// SIMATIC S7-200 SMART project (STEP 7-Micro/WIN SMART), CPU ST60

SYMBOL_TABLE Screen
X_JOG_Add_Scr    V1000.0  // X轴向上缓动按钮
X_JOG_Sub_Scr    V1000.1  // X轴向下缓动按钮
Y_JOG_Add_Scr    V1000.2
Y_JOG_Sub_Scr    V1000.3
Z_JOG_Up_Scr     V1000.4
Z_JOG_Dn_Scr     V1000.5
Teach_Btn_Setting V1000.6  // 教读设置按钮
Stop_Btn_Setting V1000.7  // 停止设置按钮
Home_Btn_Setting V1001.0  // 回原点按钮
Save_Btn_Setting V1001.1
X_Enable_Btn_Scr V1001.2
Y_Enable_Btn_Scr V1001.3
Z_Enable_Btn_Scr V1001.4
Speed_SW         V1001.5  // 速度状态指示位
Brake_Btn        V1001.6  // 刹车按钮
Clamp_Btn        V1001.7
Exit_Setting     V1005.7
Home_Lamp_Setting V1006.0  // X轴原点位指示灯
Teach_Lamp_Setting V1006.1  // 教读指示灯设置
Home_Btn_Manual  V1010.0
Stop_Btn_Manual  V1010.1
Teach_Btn_Manual V1010.2
Sholder1_Btn_Manual V1010.3
Select_Speed_Btn V1010.4  // 速度选择按钮
Sholder2_Btn_Manual V1010.5
Sholder3_Btn_Manual V1010.6
Exit_Btn_Manual  V1014.7
Home_Lamp_Manual V1015.0
Teach_Lamp_Manual V1015.1
Solder_Lamp      V1015.2
Start_Btn_Scr    V1020.0  // 屏幕运行按钮
Stop_Btn_Scr     V1020.1  // 屏幕停止按钮
Reset_Btn_Scr    V1020.2  // 复位屏幕按钮
Menu_Btn_Scr     V1020.3
Exit_MainMenu    V1020.4
Manual_Btn_Menu  V1020.5
ParaSet_Menu     V1020.6
Run_Lamp_Auto    V1021.0  // 自动运行指示灯
Stop_Lamp_Auto   V1021.1  // 自动停止指示灯
Reset_Lamp_Auto  V1021.2  // 自动复位指示灯
Run_Lamp_Blink   V1021.3
Stop_Lamp_Blink  V1021.4
Reset_Lamp_Blink V1021.5
Clr_Alarm_Btn    V1050.0
Call_Auto        V1150.0
Call_Manual      V1150.1
Call_Setting     V1150.2
Call_Solder1     V1150.3
Call_Solder2     V1150.4
Call_Solder3     V1150.5
HintTip_Stop     V1201.0  // 提示停止信息
HintTip_Reseting V1201.1  // 提示复位信息
HintTip_Running  V1201.2  // 提示运行信息
HintTip_Alarm    V1201.3  // 提示警报信息
HintTip_Ready    V1201.4  // 提示就绪信息
HintTip_Stopping V1201.5  // 提示停止信息
HintTip_Reseting1 V1201.6
X_Plus_Limit_Alarm V1501.0
X_Sub_Limit_Alarm V1501.1
Y_Plus_Limit_Alarm V1501.2
Y_Sub_Limit_Alarm V1501.3
Z_Up_Limit_Alarm V1501.4
Z_Dn_Limit_Alarm V1501.5
Clamp_At_Open_Alarm V1501.6
Clamp_At_Close_Alarm V1501.7
X_Curr_Pos_Scr   VD1900   // 屏幕X马达当前运行位置
Y_Curr_Pos_Scr   VD1904   // 屏幕Y马达当前运行位置
Z_Curr_Pos_Scr   VD1908   // 屏幕Z马达当前运行位置
X_High_Speed_Set VD4954   // X马达高速设置
X_Low_Speed_Set  VD4958   // X马达低速设置
Y_High_Speed_Set VD4962
Y_Low_Speed_Set  VD4966
Z_High_Speed_Set VD4970
Z_Low_Speed_Set  VD4974
X_Run_Speed_Set  VD4978   // X马达运行速度设置
Y_Run_Speed_Set  VD4982   // Y马达运行速度设置
Z_Run_Speed_Set  VD4986   // Z马达运行速度设置
X_POS1           VD5000
Y_POS1           VD6000
Z_POS1           VD7000
Cycle_Time       VW1100   // 单个循环周期
Choice_Aixs      VW1110
RunTip           VW1200
AlarmVar         VW1500
Screen_SW        VW1800
TotalPosNum_Set  VW4950   // 设置总的位置数值
Solder_Time      VW4952
Curr_PosNo_Scr   VW4990   // 屏幕当前XYZ马达运行位置数
Cycle_Counter    VW4992   // 循环计数器
END_SYMBOL_TABLE

SYMBOL_TABLE 系统符号
Always_On        SM0.0    // 始终接通
First_Scan_On    SM0.1    // 仅在第一个扫描周期时接通
Clock_1s         SM0.5    // 针对 1 s 的周期时间，时钟脉冲接通 0.5 s，断开 0.5 s。
P0_Config        SMB30    // 组态端口 0 通信：奇偶校验、每个字符的数据位数、波特率和协议
P0_Ctrl_Rcv      SMB87    // 接收消息控制
P0_End_Char      SMB89    // 消息结束字符
P0_Idle_Time     SMW90    // 给定的空行时间周期（以毫秒为单位）
P0_Timeout       SMW92    // 给定的字符间/消息定时器超时值（以毫秒为单位）
P0_Max_Char      SMB94    // 要接收的最大字符数（1 到 255 个字节）
END_SYMBOL_TABLE

SYMBOL_TABLE MotorStatus
X_Busy           M0.0
X_Curr_Dir       M0.1
Y_Busy           M0.2
Y_Curr_Dir       M0.3
Z_Busy           M0.4
Z_Curr_Dir       M0.5
X_Error_Code     MB1      // X马达错误代码
Y_Error_Code     MB2      // Y马达错误代码
Z_Error_Code     MB3      // Z马达运行错误代码
X_Curr_Speed     MD4      // X马达当前运行速度
Y_Curr_Speed     MD8      // Y马达当前运行速度
Z_Curr_Speed     MD12     // Z马达当前运行速度
END_SYMBOL_TABLE

SYMBOL_TABLE Machine
SpeedChoice_Pulse M18.0    // 速度选择脉冲
X_Home_EN        M18.1    // X轴归位使能信号状态位
Y_Home_EN        M18.2
Z_Home_EN        M18.3
X_Home_OK        M18.4
Y_Home_OK        M18.5
Z_Home_OK        M18.6    // Z轴准备就绪
X_Teach_EN       M18.7    // X马达教读使能
Y_Teach_EN       M19.0    // Y马达教读使能
Z_Teach_EN       M19.1    // Z马达教读使能
X_JOG_DIR        M19.2    // X轴缓动方向
Y_JOG_DIR        M19.3
Z_JOG_DIR        M19.4
X_JOG_EN         M19.5    // X轴缓动使能
Y_JOG_EN         M19.6
Z_JOG_EN         M19.7
Interlock_Manual M20.0
Interlock_Setting M20.1    // 自锁设置
X_Stop_Cmd       M20.2    // X马达停止指令
Y_Stop_Cmd       M20.3    // Y马达停止指令
Z_Stop_Cmd       M20.4    // Z马达停止指令
Motor_Ready      M20.5    // 马达就绪
XYZ_ORG_Cmd3     M22.0
XYZ_Home_OK      M20.6    // XYZ归位信号状态位
Z_Goto_UpPos     M20.7    // Z轴上升到最高位信号状态位
Init_MC_Sys      M21.0
XYZ_ORG_Cmd1     M21.6
XYZ_ORG_Cmd      M21.1    // XYZ归位起始位指令
Release_Brake_Step M21.2
Solder2_Cmd      M21.4
Solder3_Cmd      M21.5
Solder1_Cmd      M21.3
Step1_Auto_Lock  M25.0    // 自动锁定step1
Step1_Auto       M25.1    // 自动step1
Step2_X_Auto     M25.2    // X轴自动step2
Step2_Y_Auto     M25.3    // Y轴自动step2
Step3_Auto       M25.4    // 自动step3
Step4_Auto       M25.5    // 自动step4
X_Cmd_Pos        VD2000   // X马达位置指令
Y_Cmd_Pos        VD2004   // Y马达位置指令
Z_Cmd_Pos        VD2008   // Z马达位置指令
X_Debug_Speed    VD2012   // X马达调试（运行）速度
Y_Debug_Speed    VD2016
Z_Debug_Speed    VD2020   // Z马达调试速度
Cycle_Timer      T50      // 循环计时器
Sholder_Timer    T35
Solder_timer     T36
Brake_Release_Timer T34
Z_Home2          M29.2
Z_Home3          M29.3
Z_Home1          M29.1
XYZ_ORG_Cmd2     M21.7
END_SYMBOL_TABLE

SYMBOL_TABLE INPUT
X_AXIS_ZP        I0.0     // X轴马达索引
Y_AXIS_ZP        I0.1     // Y轴马达索引
Z_AXIS_ZP        I0.2     // Z轴马达索引
X_AXIS_LMT_Plus  I0.3     // X轴马达正限
X_AXIS_LMT_Sub   I0.4     // X轴马达负限
X_AXIS_HOME      I0.5     // X轴马达原点
Y_AXIS_LMT_Plus  I0.6     // Y轴马达正限
Y_AXIS_LMT_Sub   I0.7     // Y轴马达负限
Y_AXIS_HOME      I1.0     // Y轴马达原点
Z_AXIS_LMT_Plus  I1.1     // Z轴马达正限
Z_AXIS_LMT_Sub   I1.2     // Z轴马达负限
Z_AXIS_HOME      I1.3     // Z轴马达原点
X_AXIS_INPOS     I1.4     // X轴位置完成
X_AXIS_READY     I1.5     // X轴准备信号
X_AXIS_ALARM     I1.6     // X轴报警信号
Y_AXIS_INPOS     I1.7     // Y轴位置完成
Y_AXIS_READY     I2.0     // Y轴准备信号
Y_AXIS_ALARM     I2.1     // Y轴报警信号
Z_AXIS_INPOS     I2.2     // Z轴位置完成
Z_AXIS_READY     I2.3     // Z轴准备信号
Z_AXIS_ALARM     I2.4     // Z轴报警信号
START_BUTTON     I2.5     // 启动按钮
STOP_BUTTON      I2.6     // 停止按钮
RESET_BUTTON     I2.7     // 复位按钮
CLAMP_AT_OPEN    I3.0     // 夹子打开感应
CLAMP_AT_CLOSE   I3.1     // 夹子关闭感应
END_SYMBOL_TABLE

SYMBOL_TABLE OUTPUT
X_AXIS_PULSE     Q0.0     // X轴脉冲信号
Y_AXIS_PULSE     Q0.1     // Y轴脉冲信号
X_AXIS_DIR       Q0.2     // X轴方向信号
Z_AXIS_PULSE     Q0.3     // Z轴脉冲信号
X_AXIS_ENABLE    Q0.4     // X轴使能信号
Y_AXIS_ENABLE    Q0.5     // Y轴使能信号
Z_AXIS_ENABLE    Q0.6     // Z轴使能信号
Y_AXIS_DIR       Q0.7     // Y轴方向信号
Z_AXIS_DIR       Q1.0     // Z轴方向信号
X_ALARM_CLEAR    Q1.1     // X轴报警清除
Y_ALARM_CLEAR    Q1.2     // Y轴报警清除
Z_ALARM_CLEAR    Q1.3     // Z轴报警清除
Z_BRAKE_RELEASE  Q1.4     // Z轴刹车释放
CLAMP_OPEN_VALVE Q1.5     // 夹打开阀
CLAMP_CLOSE_VALVE Q1.6     // 夹关闭阀
START_LAMP       Q2.0     // 启动指示灯
STOP_LAMP        Q2.1     // 停止指示灯
RESET_LAMP       Q2.2     // 复位指示灯
END_SYMBOL_TABLE

SYMBOL_TABLE Solder1
Step1_Solder1    M26.0
Step2_Solder1    M26.1
Step3_Solder1    M26.2
Step4_Solder1    M26.3
Step5_Solder1    M26.4
Step6_Solder1    M26.5
Step7_Solder1    M26.6
X_No_1           VD3000
X_No_2           VD3004
solder_No1       VW4998
END_SYMBOL_TABLE

SYMBOL_TABLE Solder3
Step1_Solder3    M27.3
Step2_Solder3    M27.4
Step3_Solder3    M27.5
Step4_Solder3    M27.6
Step5_Solder3    M27.7
Step6_Solder3    M28.0
Step7_Solder3    M28.1
Step8_Solder3    M28.2
END_SYMBOL_TABLE

SYMBOL_TABLE Solder2
Step1_Solder2    M28.3
Step2_Solder2    M28.4
Step3_Solder2    M26.7
Step4_Solder2    M27.0
Step5_Solder2    M27.1
Step6_Solder2    M27.2
Step7_Solder2    M28.5
Step8_Solder2    M28.6
END_SYMBOL_TABLE

ORGANIZATION_BLOCK 程序块:OB1
TITLE=程序注释
VAR
AutoScreen:WORD;	// LW0 
ManualScreen:WORD;	// LW2 
SettingScreen:WORD;	// LW4 
AlarmScreen:WORD;	// LW6 
MainScreen:WORD;	// LW8 
END_VAR
BEGIN
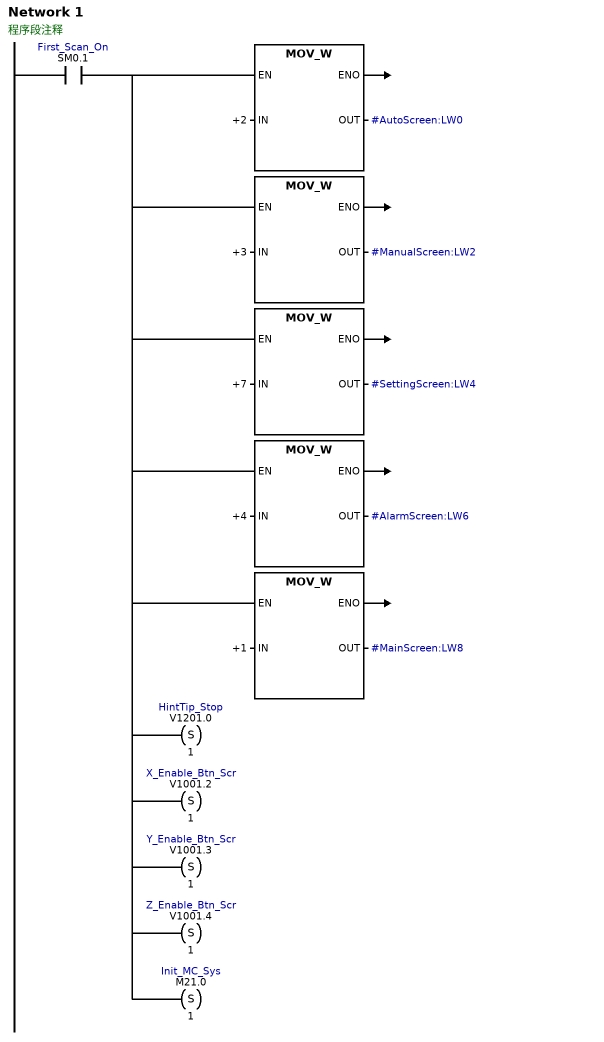
Network 1
// 程序段注释
LD     First_Scan_On:SM0.1
MOVW   +2, #AutoScreen:LW0
MOVW   +3, #ManualScreen:LW2
MOVW   +7, #SettingScreen:LW4
MOVW   +4, #AlarmScreen:LW6
MOVW   +1, #MainScreen:LW8
S      HintTip_Stop:V1201.0, 1
S      X_Enable_Btn_Scr:V1001.2, 1
S      Y_Enable_Btn_Scr:V1001.3, 1
S      Z_Enable_Btn_Scr:V1001.4, 1
S      Init_MC_Sys:M21.0, 1
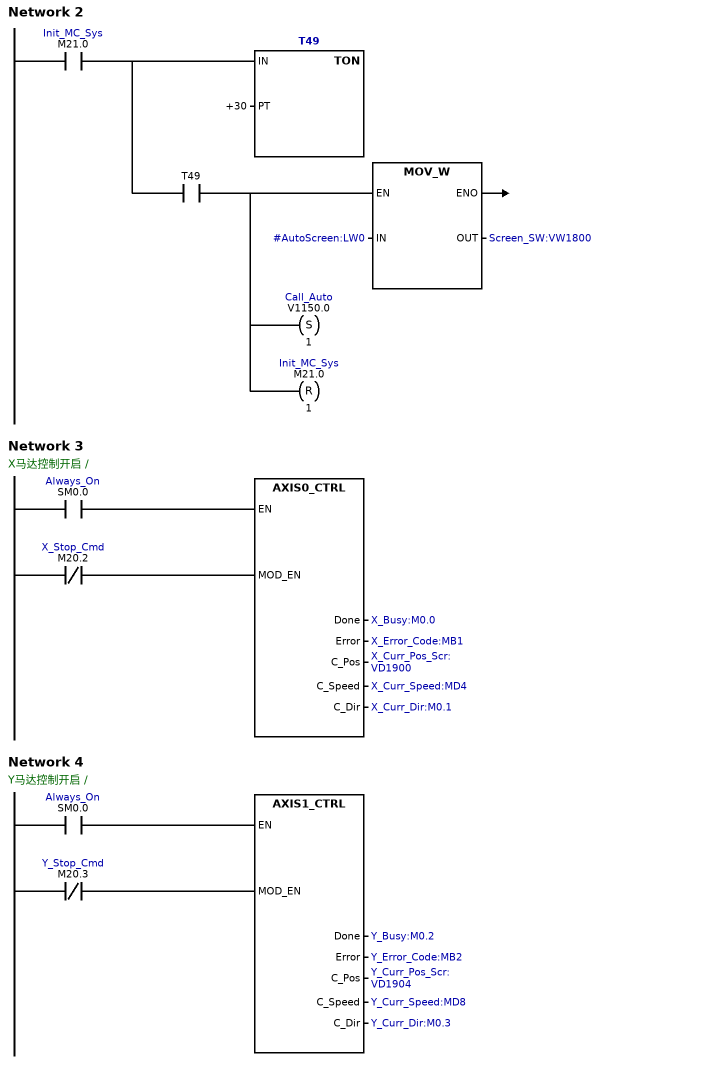
Network 2
LD     Init_MC_Sys:M21.0
TON    T49, +30
A      T49
MOVW   #AutoScreen:LW0, Screen_SW:VW1800
S      Call_Auto:V1150.0, 1
R      Init_MC_Sys:M21.0, 1
Network 3
// X马达控制开启
// 
LD     Always_On:SM0.0
=      L60.0
LDN    X_Stop_Cmd:M20.2
=      L63.7
LD     L60.0
CALL   AXIS0_CTRL:SBR1, L63.7, X_Busy:M0.0, X_Error_Code:MB1, X_Curr_Pos_Scr:VD1900, X_Curr_Speed:MD4, X_Curr_Dir:M0.1
Network 4
// Y马达控制开启
// 
LD     Always_On:SM0.0
=      L60.0
LDN    Y_Stop_Cmd:M20.3
=      L63.7
LD     L60.0
CALL   AXIS1_CTRL:SBR12, L63.7, Y_Busy:M0.2, Y_Error_Code:MB2, Y_Curr_Pos_Scr:VD1904, Y_Curr_Speed:MD8, Y_Curr_Dir:M0.3
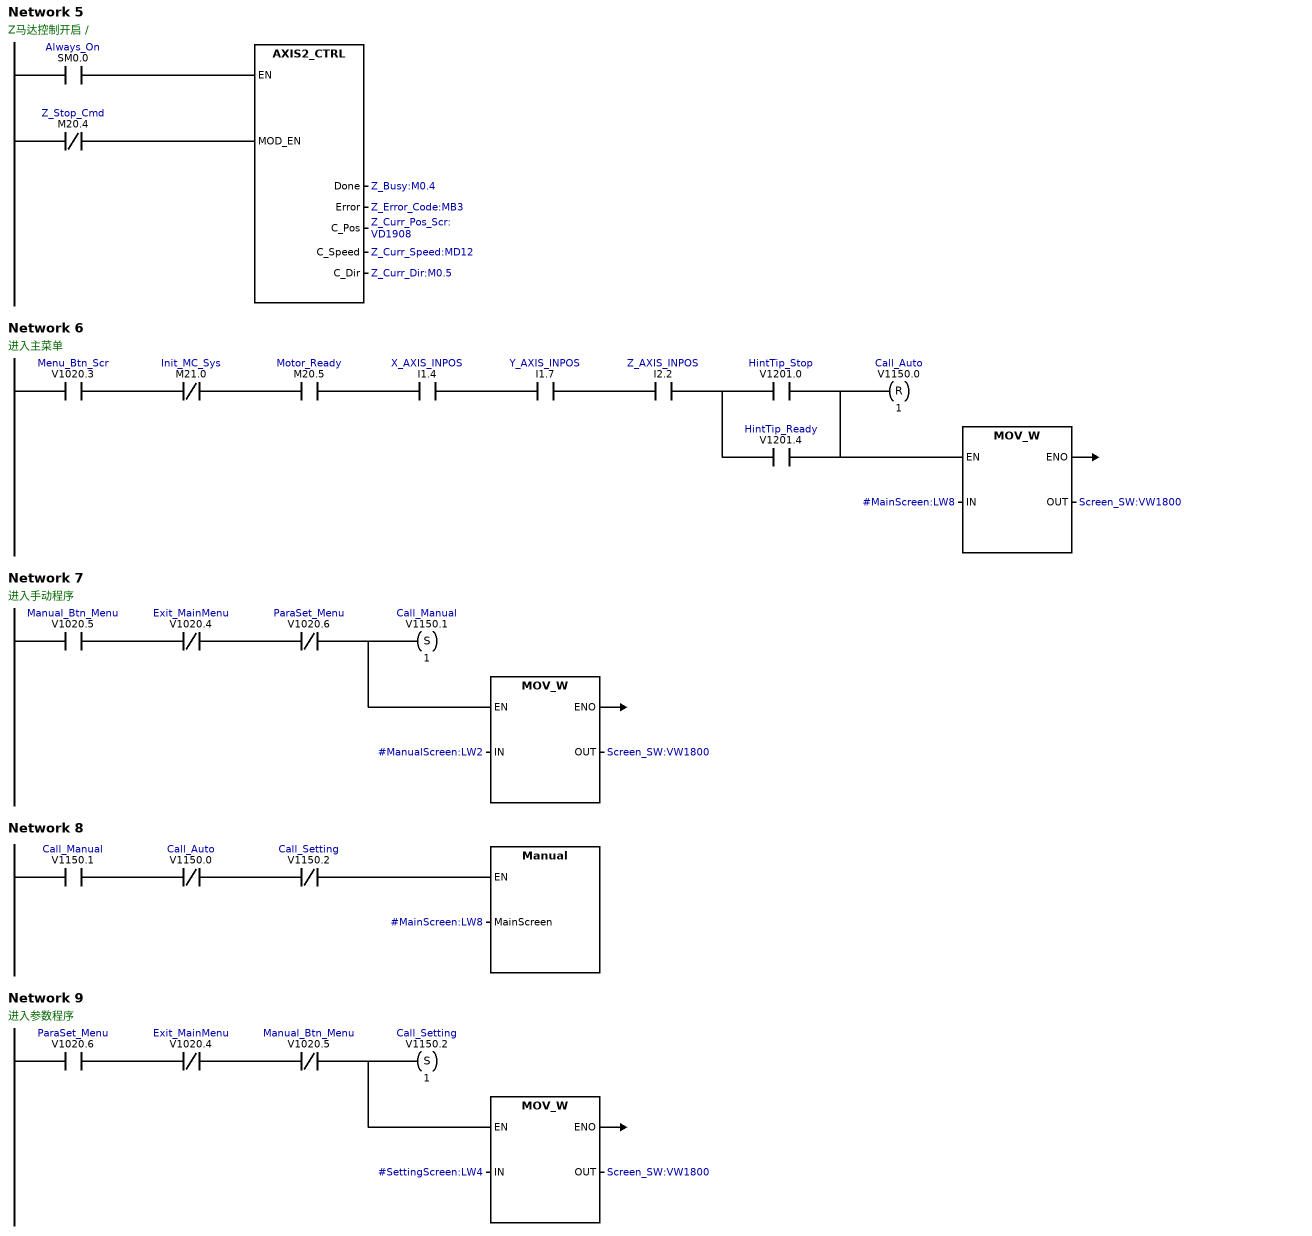
Network 5
// Z马达控制开启
// 
LD     Always_On:SM0.0
=      L60.0
LDN    Z_Stop_Cmd:M20.4
=      L63.7
LD     L60.0
CALL   AXIS2_CTRL:SBR23, L63.7, Z_Busy:M0.4, Z_Error_Code:MB3, Z_Curr_Pos_Scr:VD1908, Z_Curr_Speed:MD12, Z_Curr_Dir:M0.5
Network 6
// 进入主菜单
LD     Menu_Btn_Scr:V1020.3
AN     Init_MC_Sys:M21.0
A      Motor_Ready:M20.5
A      X_AXIS_INPOS:I1.4
A      Y_AXIS_INPOS:I1.7
A      Z_AXIS_INPOS:I2.2
LD     HintTip_Stop:V1201.0
O      HintTip_Ready:V1201.4
ALD
R      Call_Auto:V1150.0, 1
MOVW   #MainScreen:LW8, Screen_SW:VW1800
Network 7
// 进入手动程序
LD     Manual_Btn_Menu:V1020.5
AN     Exit_MainMenu:V1020.4
AN     ParaSet_Menu:V1020.6
S      Call_Manual:V1150.1, 1
MOVW   #ManualScreen:LW2, Screen_SW:VW1800
Network 8
LD     Call_Manual:V1150.1
AN     Call_Auto:V1150.0
AN     Call_Setting:V1150.2
CALL   Manual:SBR0, #MainScreen:LW8
Network 9
// 进入参数程序
LD     ParaSet_Menu:V1020.6
AN     Exit_MainMenu:V1020.4
AN     Manual_Btn_Menu:V1020.5
S      Call_Setting:V1150.2, 1
MOVW   #SettingScreen:LW4, Screen_SW:VW1800
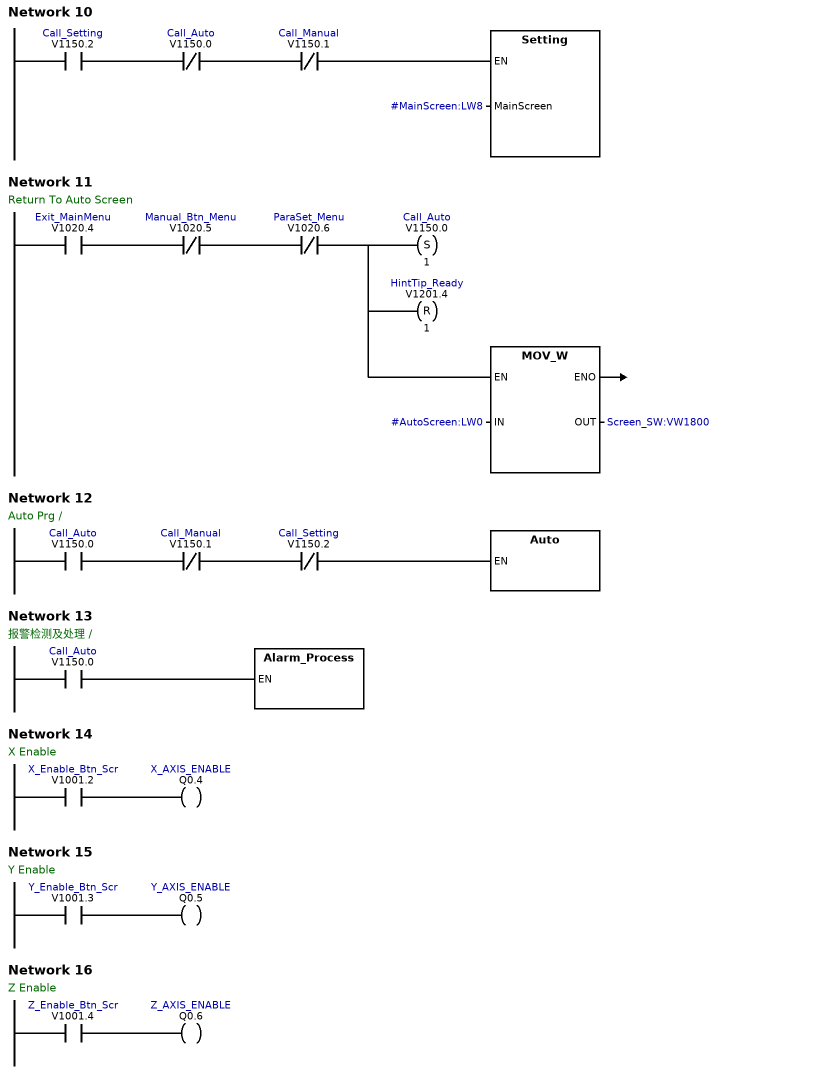
Network 10
LD     Call_Setting:V1150.2
AN     Call_Auto:V1150.0
AN     Call_Manual:V1150.1
CALL   Setting:SBR35, #MainScreen:LW8
Network 11
// Return To Auto Screen
LD     Exit_MainMenu:V1020.4
AN     Manual_Btn_Menu:V1020.5
AN     ParaSet_Menu:V1020.6
S      Call_Auto:V1150.0, 1
R      HintTip_Ready:V1201.4, 1
MOVW   #AutoScreen:LW0, Screen_SW:VW1800
Network 12
// Auto Prg
// 
LD     Call_Auto:V1150.0
AN     Call_Manual:V1150.1
AN     Call_Setting:V1150.2
CALL   Auto:SBR34
Network 13
// 报警检测及处理
// 
LD     Call_Auto:V1150.0
CALL   Alarm_Process:SBR36
Network 14
// X Enable
LD     X_Enable_Btn_Scr:V1001.2
=      X_AXIS_ENABLE:Q0.4
Network 15
// Y Enable
LD     Y_Enable_Btn_Scr:V1001.3
=      Y_AXIS_ENABLE:Q0.5
Network 16
// Z Enable
LD     Z_Enable_Btn_Scr:V1001.4
=      Z_AXIS_ENABLE:Q0.6
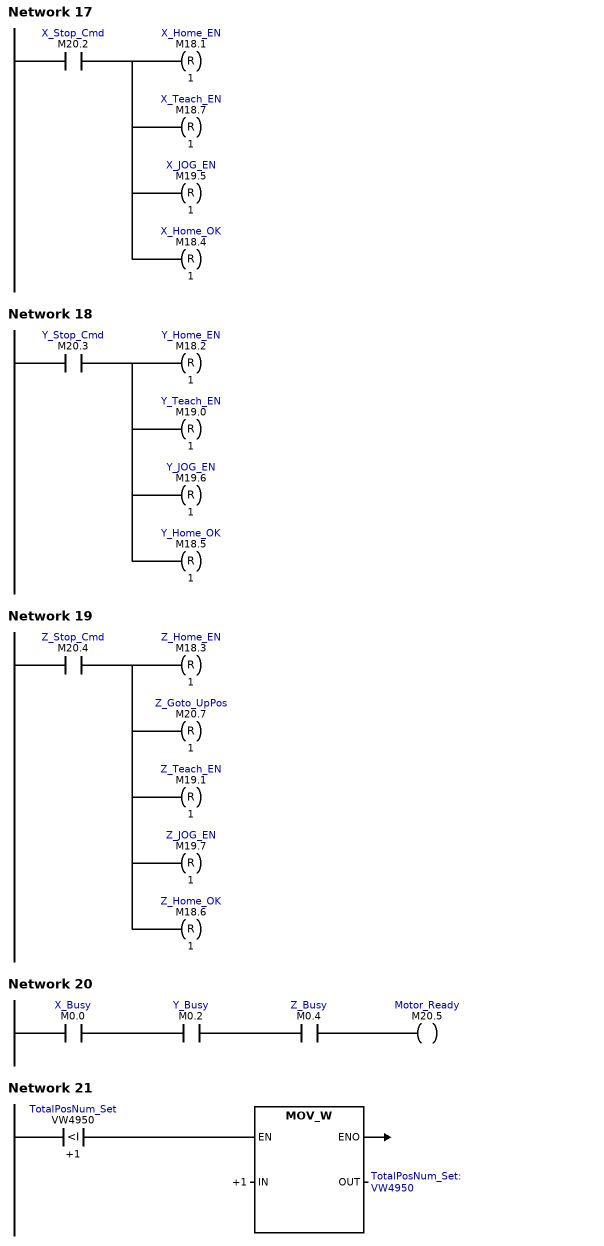
Network 17
LD     X_Stop_Cmd:M20.2
R      X_Home_EN:M18.1, 1
R      X_Teach_EN:M18.7, 1
R      X_JOG_EN:M19.5, 1
R      X_Home_OK:M18.4, 1
Network 18
LD     Y_Stop_Cmd:M20.3
R      Y_Home_EN:M18.2, 1
R      Y_Teach_EN:M19.0, 1
R      Y_JOG_EN:M19.6, 1
R      Y_Home_OK:M18.5, 1
Network 19
LD     Z_Stop_Cmd:M20.4
R      Z_Home_EN:M18.3, 1
R      Z_Goto_UpPos:M20.7, 1
R      Z_Teach_EN:M19.1, 1
R      Z_JOG_EN:M19.7, 1
R      Z_Home_OK:M18.6, 1
Network 20
LD     X_Busy:M0.0
A      Y_Busy:M0.2
A      Z_Busy:M0.4
=      Motor_Ready:M20.5
Network 21
LDW<   TotalPosNum_Set:VW4950, +1
MOVW   +1, TotalPosNum_Set:VW4950
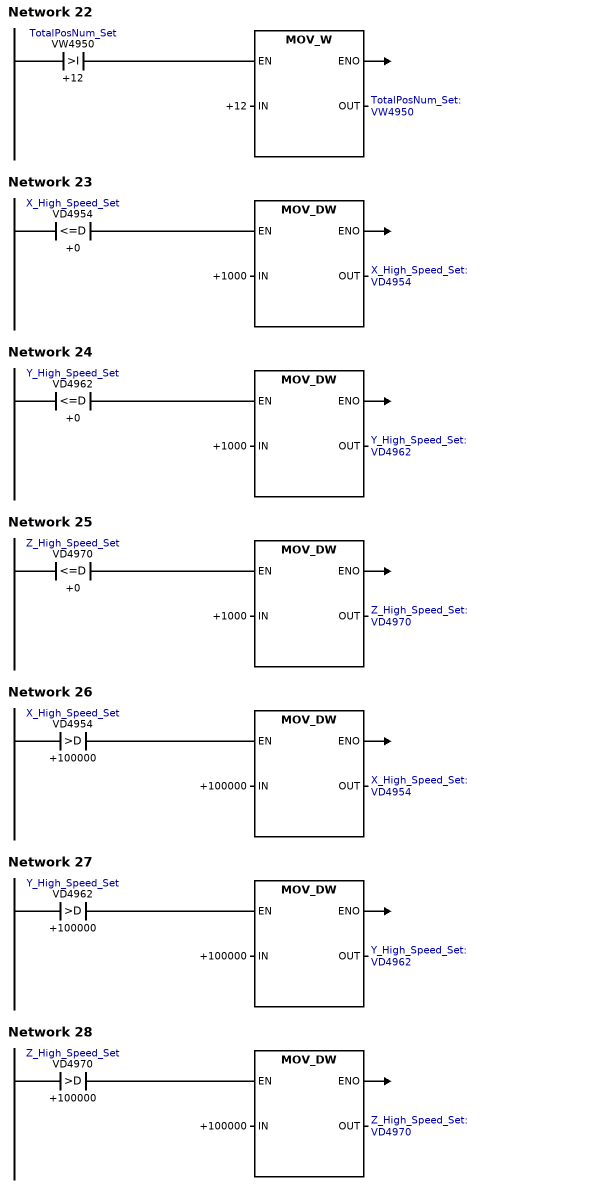
Network 22
LDW>   TotalPosNum_Set:VW4950, +12
MOVW   +12, TotalPosNum_Set:VW4950
Network 23
LDD<=  X_High_Speed_Set:VD4954, +0
MOVD   +1000, X_High_Speed_Set:VD4954
Network 24
LDD<=  Y_High_Speed_Set:VD4962, +0
MOVD   +1000, Y_High_Speed_Set:VD4962
Network 25
LDD<=  Z_High_Speed_Set:VD4970, +0
MOVD   +1000, Z_High_Speed_Set:VD4970
Network 26
LDD>   X_High_Speed_Set:VD4954, +100000
MOVD   +100000, X_High_Speed_Set:VD4954
Network 27
LDD>   Y_High_Speed_Set:VD4962, +100000
MOVD   +100000, Y_High_Speed_Set:VD4962
Network 28
LDD>   Z_High_Speed_Set:VD4970, +100000
MOVD   +100000, Z_High_Speed_Set:VD4970
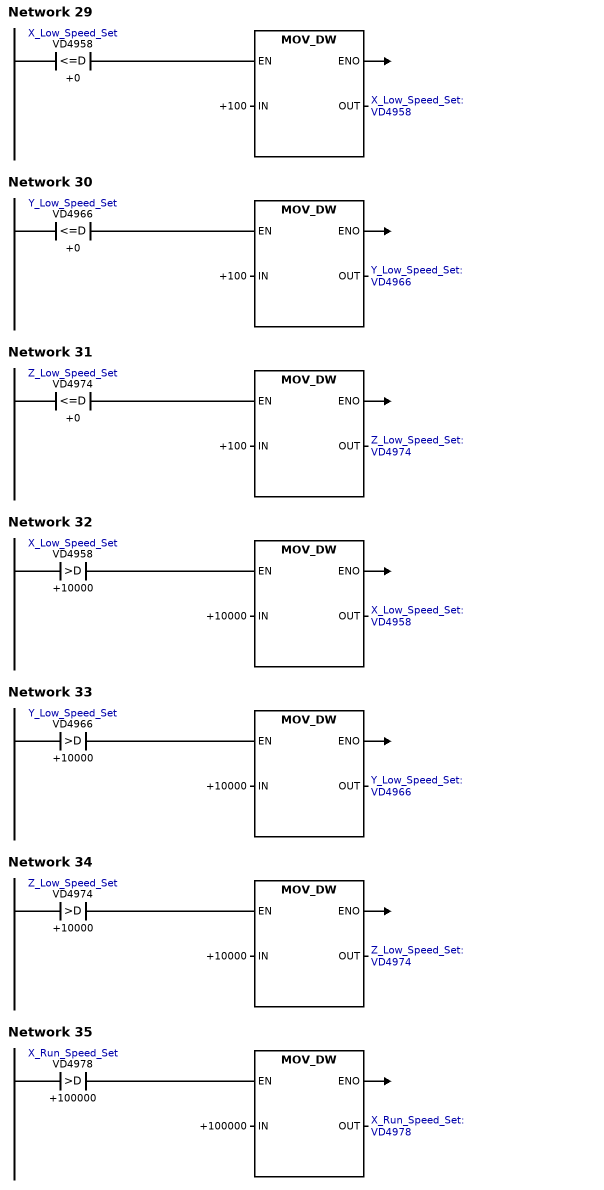
Network 29
LDD<=  X_Low_Speed_Set:VD4958, +0
MOVD   +100, X_Low_Speed_Set:VD4958
Network 30
LDD<=  Y_Low_Speed_Set:VD4966, +0
MOVD   +100, Y_Low_Speed_Set:VD4966
Network 31
LDD<=  Z_Low_Speed_Set:VD4974, +0
MOVD   +100, Z_Low_Speed_Set:VD4974
Network 32
LDD>   X_Low_Speed_Set:VD4958, +10000
MOVD   +10000, X_Low_Speed_Set:VD4958
Network 33
LDD>   Y_Low_Speed_Set:VD4966, +10000
MOVD   +10000, Y_Low_Speed_Set:VD4966
Network 34
LDD>   Z_Low_Speed_Set:VD4974, +10000
MOVD   +10000, Z_Low_Speed_Set:VD4974
Network 35
LDD>   X_Run_Speed_Set:VD4978, +100000
MOVD   +100000, X_Run_Speed_Set:VD4978
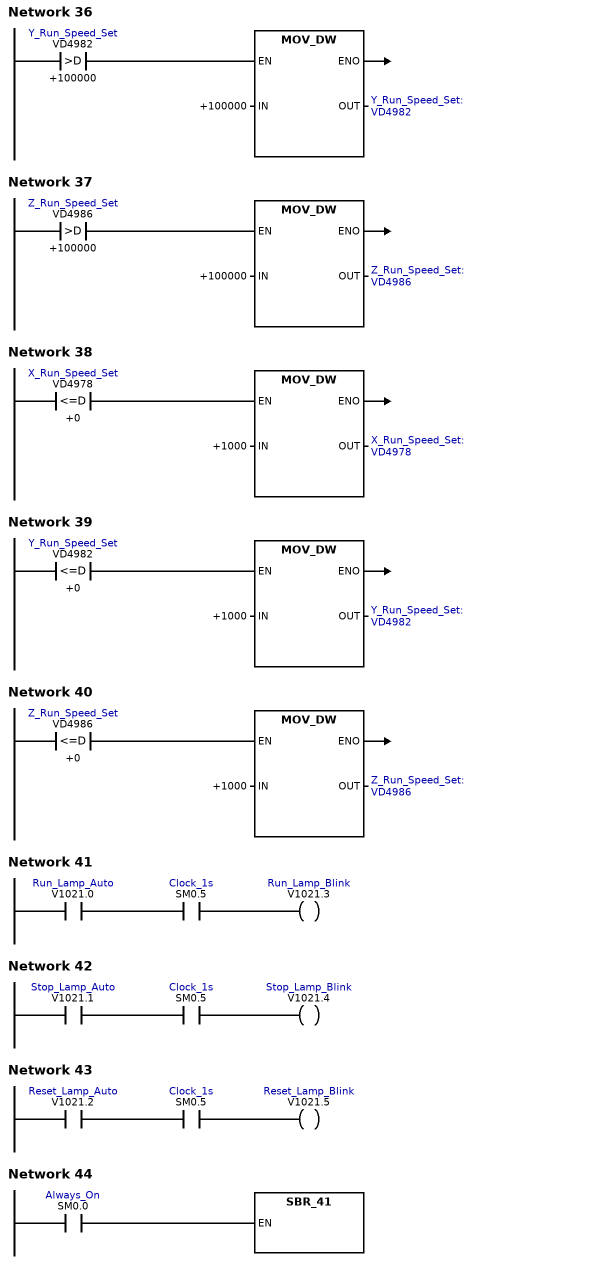
Network 36
LDD>   Y_Run_Speed_Set:VD4982, +100000
MOVD   +100000, Y_Run_Speed_Set:VD4982
Network 37
LDD>   Z_Run_Speed_Set:VD4986, +100000
MOVD   +100000, Z_Run_Speed_Set:VD4986
Network 38
LDD<=  X_Run_Speed_Set:VD4978, +0
MOVD   +1000, X_Run_Speed_Set:VD4978
Network 39
LDD<=  Y_Run_Speed_Set:VD4982, +0
MOVD   +1000, Y_Run_Speed_Set:VD4982
Network 40
LDD<=  Z_Run_Speed_Set:VD4986, +0
MOVD   +1000, Z_Run_Speed_Set:VD4986
Network 41
LD     Run_Lamp_Auto:V1021.0
A      Clock_1s:SM0.5
=      Run_Lamp_Blink:V1021.3
Network 42
LD     Stop_Lamp_Auto:V1021.1
A      Clock_1s:SM0.5
=      Stop_Lamp_Blink:V1021.4
Network 43
LD     Reset_Lamp_Auto:V1021.2
A      Clock_1s:SM0.5
=      Reset_Lamp_Blink:V1021.5
Network 44
LD     Always_On:SM0.0
CALL   SBR_41:SBR41
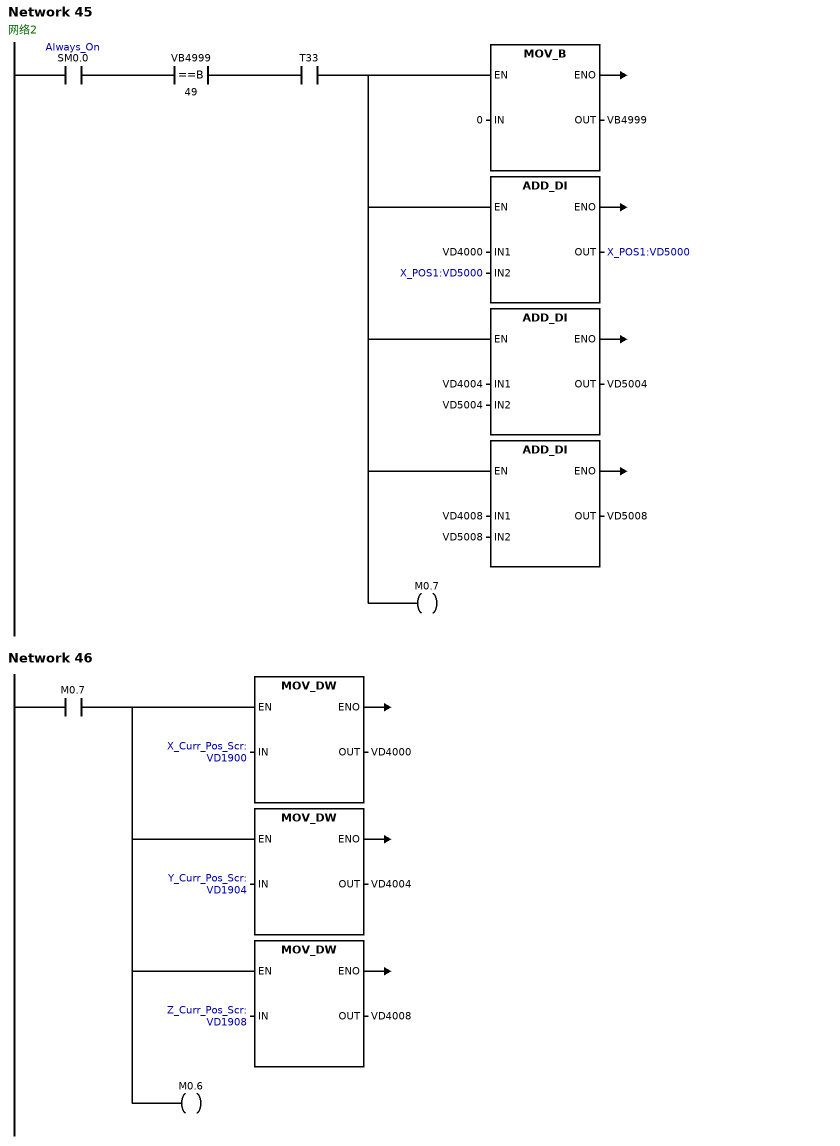
Network 45
// 网络2  
LD     Always_On:SM0.0
AB=    VB4999, 49
A      T33
MOVB   0, VB4999
+D     VD4000, X_POS1:VD5000
+D     VD4004, VD5004
+D     VD4008, VD5008
=      M0.7
Network 46
//   
LD     M0.7
MOVD   X_Curr_Pos_Scr:VD1900, VD4000
MOVD   Y_Curr_Pos_Scr:VD1904, VD4004
MOVD   Z_Curr_Pos_Scr:VD1908, VD4008
=      M0.6
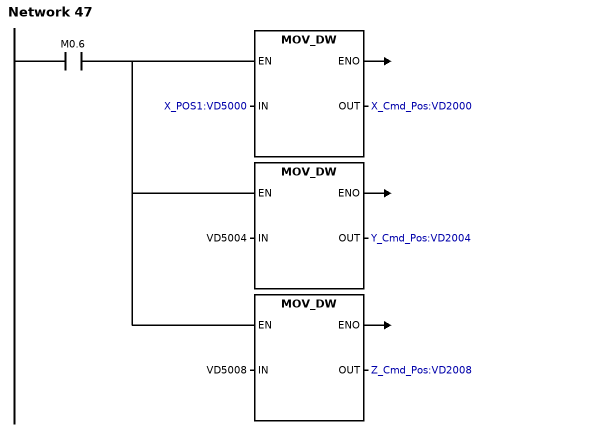
Network 47
LD     M0.6
MOVD   X_POS1:VD5000, X_Cmd_Pos:VD2000
MOVD   VD5004, Y_Cmd_Pos:VD2004
MOVD   VD5008, Z_Cmd_Pos:VD2008
END_ORGANIZATION_BLOCK

SUBROUTINE_BLOCK Manual:SBR0
TITLE=子例程注释
VAR_INPUT
MainScreen:WORD;	// LW0 
END_VAR
VAR
X_Home_Err:BYTE;	// LB2 
Y_Home_Err:BYTE;	// LB3 
Z_Home_Err:BYTE;	// LB4 
X_Teach_Done:BOOL;	// L5.0 
Y_Teach_Done:BOOL;	// L5.1 
Z_Teach_Done:BOOL;	// L5.2 
X_Teach_Err:BYTE;	// LB6 
Y_Teach_Err:BYTE;	// LB7 
Z_Teach_Err:BYTE;	// LB8 
X_JOG_ERR:BYTE;	// LB9 
Y_JOG_ERR:BYTE;	// LB10 
Z_JOG_ERR:BYTE;	// LB11 
X_Curr_Dir:BOOL;	// L12.0 
Y_Curr_Dir:BOOL;	// L12.1 
Z_Curr_Dir:BOOL;	// L12.2 
END_VAR
BEGIN
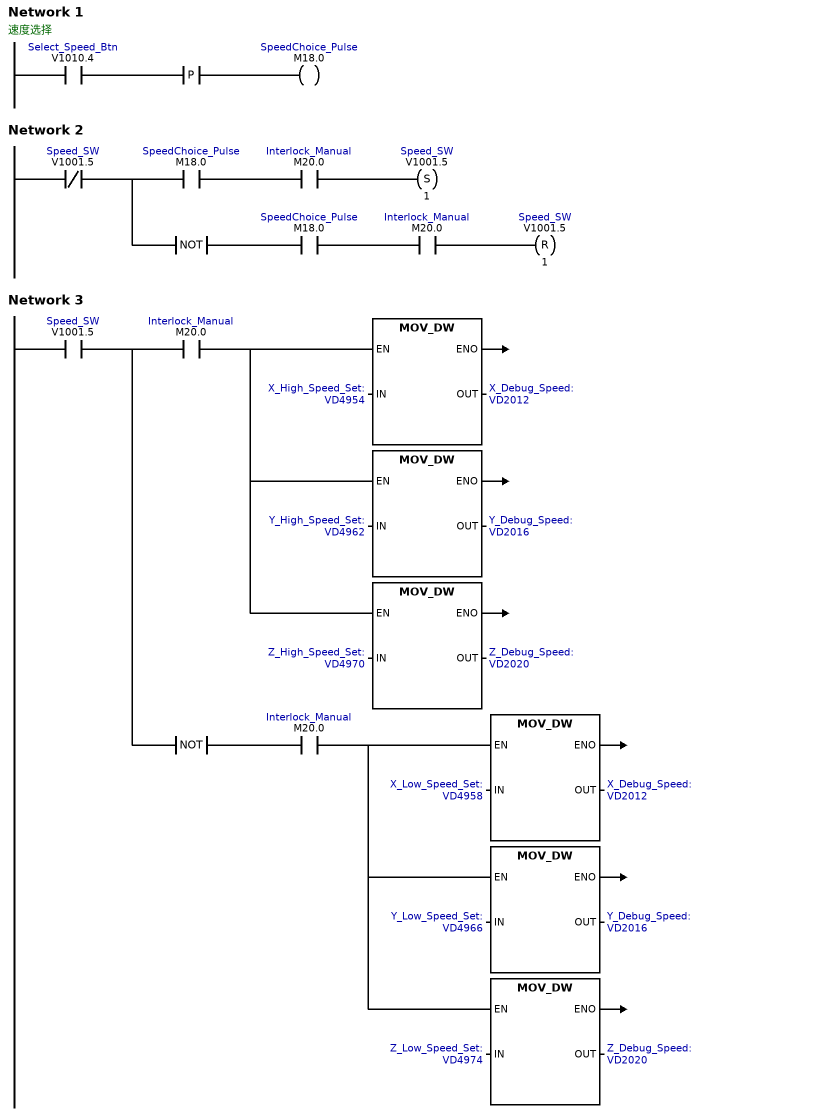
Network 1
// 速度选择
LD     Select_Speed_Btn:V1010.4
EU
=      SpeedChoice_Pulse:M18.0
Network 2
LDN    Speed_SW:V1001.5
LPS
A      SpeedChoice_Pulse:M18.0
A      Interlock_Manual:M20.0
S      Speed_SW:V1001.5, 1
LPP
NOT
A      SpeedChoice_Pulse:M18.0
A      Interlock_Manual:M20.0
R      Speed_SW:V1001.5, 1
Network 3
LD     Speed_SW:V1001.5
LPS
A      Interlock_Manual:M20.0
MOVD   X_High_Speed_Set:VD4954, X_Debug_Speed:VD2012
MOVD   Y_High_Speed_Set:VD4962, Y_Debug_Speed:VD2016
MOVD   Z_High_Speed_Set:VD4970, Z_Debug_Speed:VD2020
LPP
NOT
A      Interlock_Manual:M20.0
MOVD   X_Low_Speed_Set:VD4958, X_Debug_Speed:VD2012
MOVD   Y_Low_Speed_Set:VD4966, Y_Debug_Speed:VD2016
MOVD   Z_Low_Speed_Set:VD4974, Z_Debug_Speed:VD2020
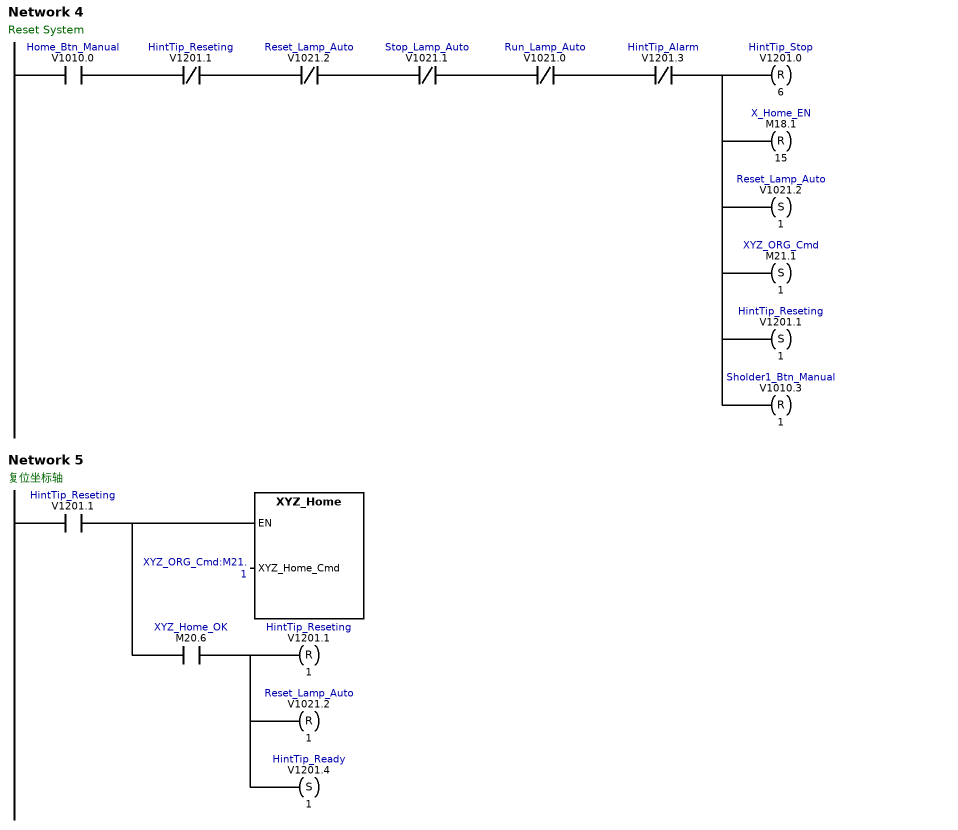
Network 4
// Reset System
LD     Home_Btn_Manual:V1010.0
AN     HintTip_Reseting:V1201.1
AN     Reset_Lamp_Auto:V1021.2
AN     Stop_Lamp_Auto:V1021.1
AN     Run_Lamp_Auto:V1021.0
AN     HintTip_Alarm:V1201.3
R      HintTip_Stop:V1201.0, 6
R      X_Home_EN:M18.1, 15
S      Reset_Lamp_Auto:V1021.2, 1
S      XYZ_ORG_Cmd:M21.1, 1
S      HintTip_Reseting:V1201.1, 1
R      Sholder1_Btn_Manual:V1010.3, 1
Network 5
// 复位坐标轴
LD     HintTip_Reseting:V1201.1
CALL   XYZ_Home:SBR37, XYZ_ORG_Cmd:M21.1
A      XYZ_Home_OK:M20.6
R      HintTip_Reseting:V1201.1, 1
R      Reset_Lamp_Auto:V1021.2, 1
S      HintTip_Ready:V1201.4, 1
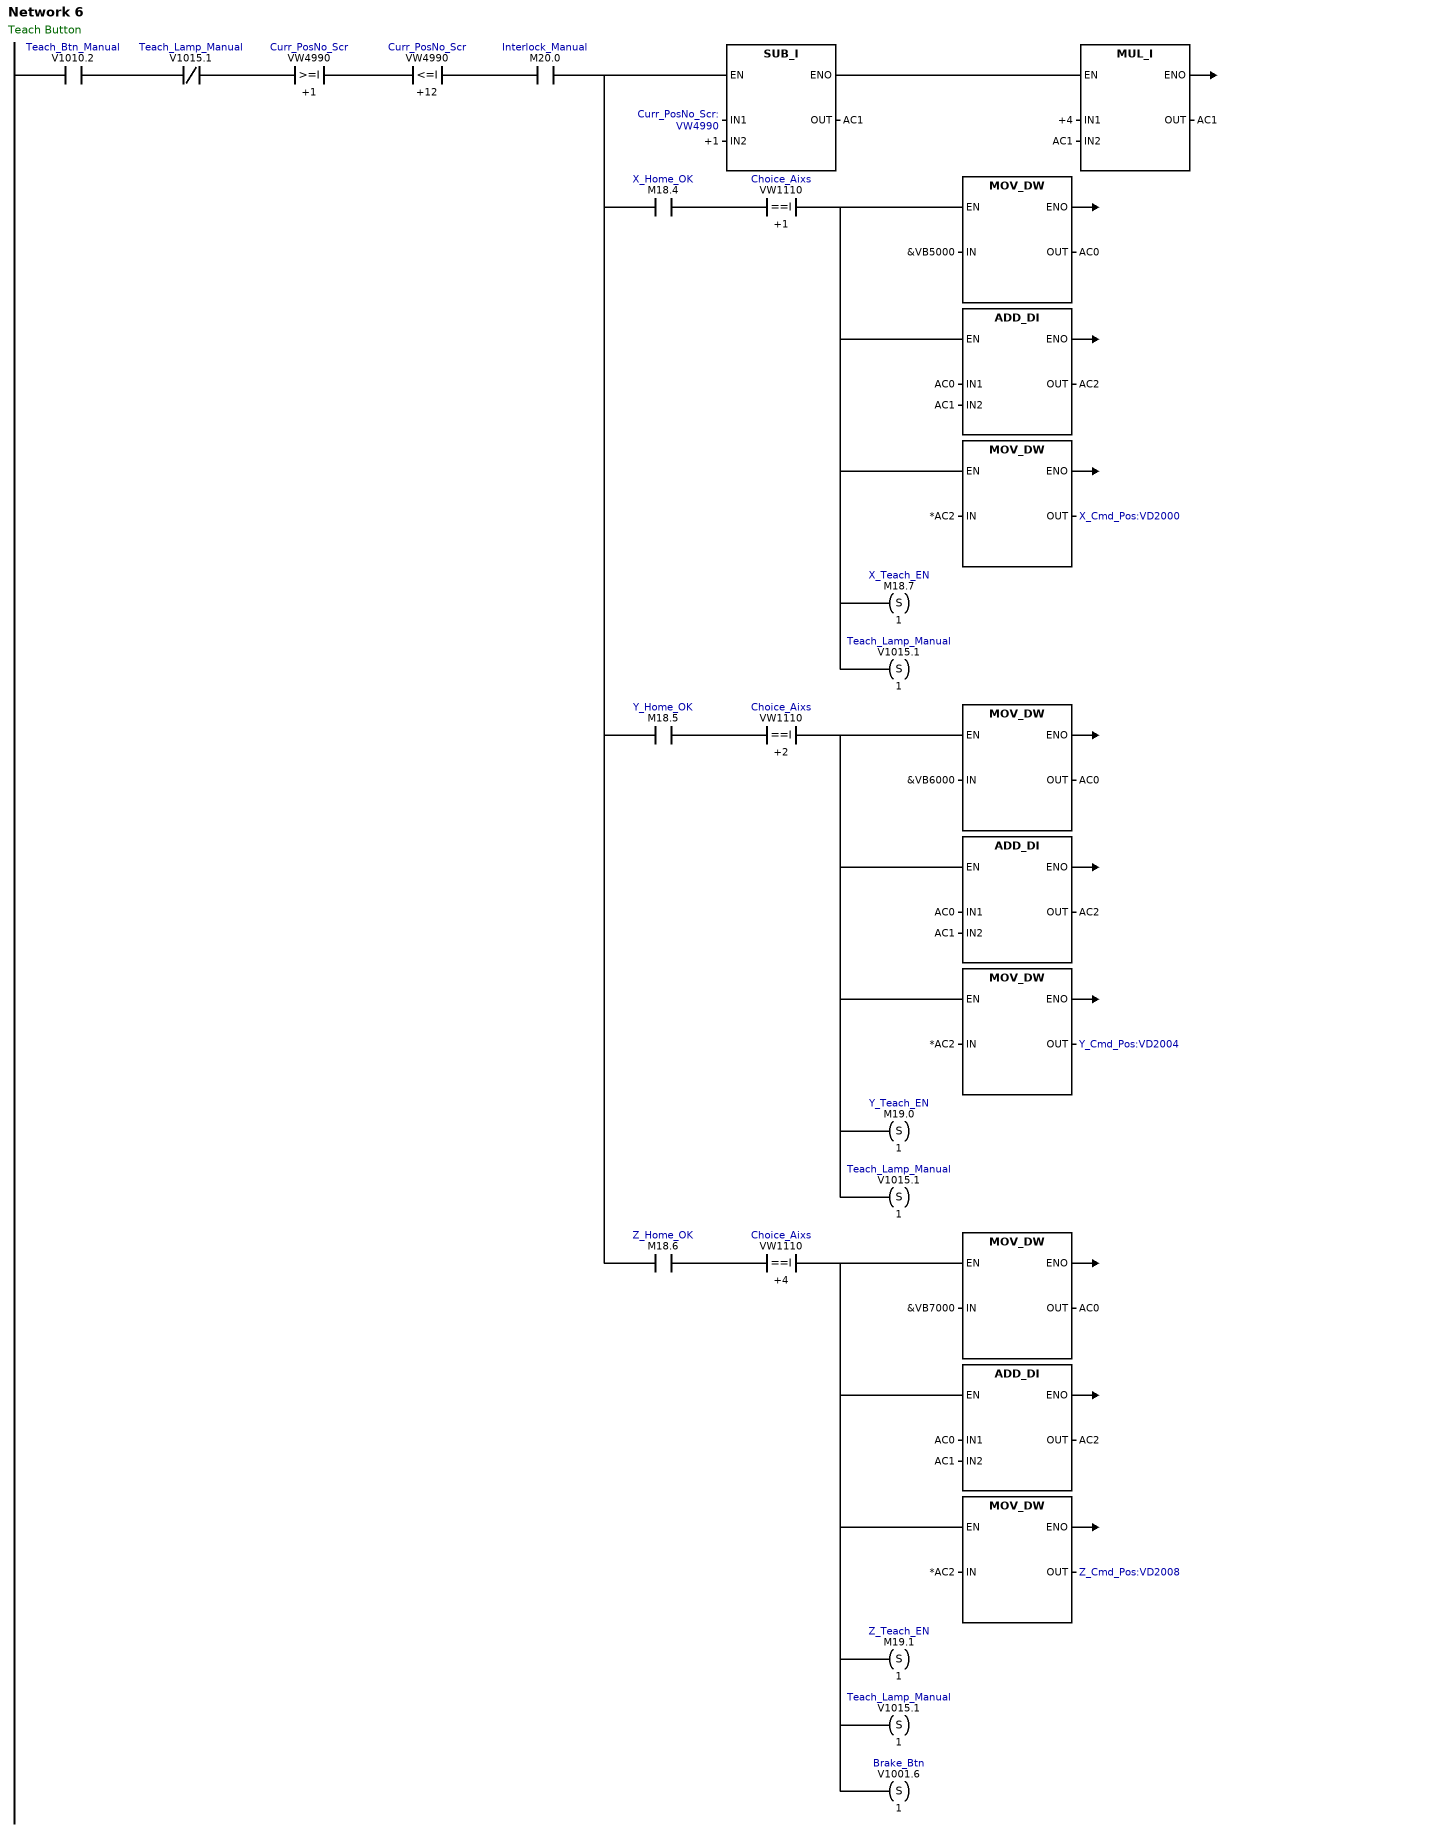
Network 6
// Teach Button
LD     Teach_Btn_Manual:V1010.2
AN     Teach_Lamp_Manual:V1015.1
AW>=   Curr_PosNo_Scr:VW4990, +1
AW<=   Curr_PosNo_Scr:VW4990, +12
A      Interlock_Manual:M20.0
LPS
MOVW   Curr_PosNo_Scr:VW4990, AC1
AENO
-I     +1, AC1
AENO
*I     +4, AC1
LRD
A      X_Home_OK:M18.4
AW=    Choice_Aixs:VW1110, +1
MOVD   &VB5000, AC0
MOVD   AC0, AC2
+D     AC1, AC2
MOVD   *AC2, X_Cmd_Pos:VD2000
S      X_Teach_EN:M18.7, 1
S      Teach_Lamp_Manual:V1015.1, 1
LRD
A      Y_Home_OK:M18.5
AW=    Choice_Aixs:VW1110, +2
MOVD   &VB6000, AC0
MOVD   AC0, AC2
+D     AC1, AC2
MOVD   *AC2, Y_Cmd_Pos:VD2004
S      Y_Teach_EN:M19.0, 1
S      Teach_Lamp_Manual:V1015.1, 1
LPP
A      Z_Home_OK:M18.6
AW=    Choice_Aixs:VW1110, +4
MOVD   &VB7000, AC0
MOVD   AC0, AC2
+D     AC1, AC2
MOVD   *AC2, Z_Cmd_Pos:VD2008
S      Z_Teach_EN:M19.1, 1
S      Teach_Lamp_Manual:V1015.1, 1
S      Brake_Btn:V1001.6, 1
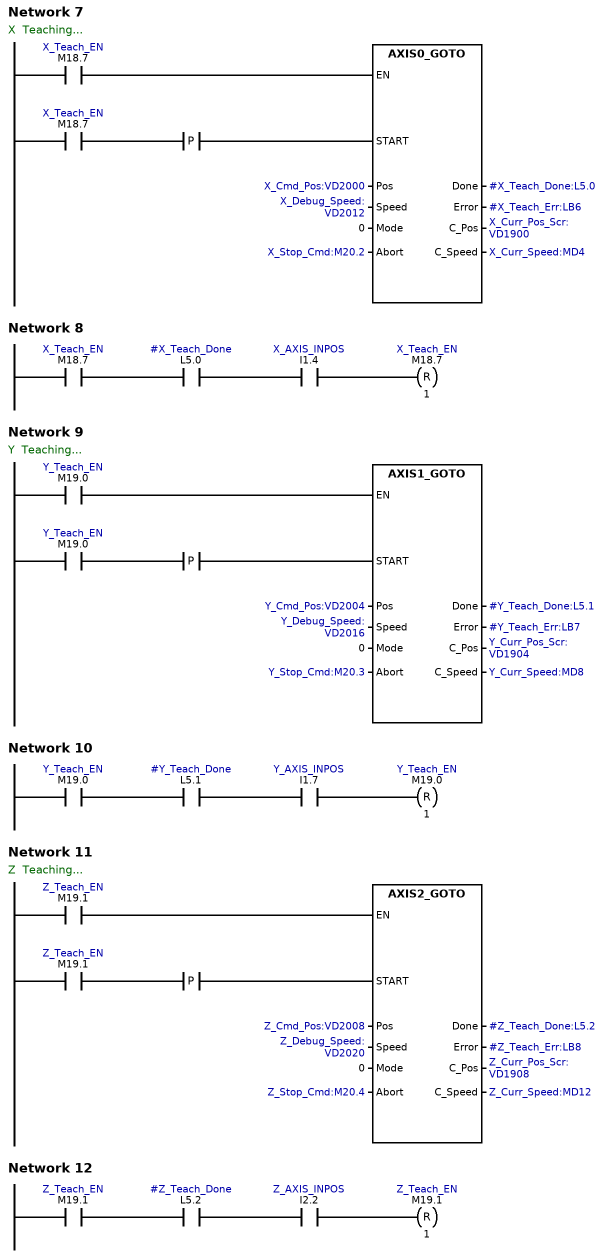
Network 7
// X  Teaching...
LD     X_Teach_EN:M18.7
=      L60.0
LD     X_Teach_EN:M18.7
EU
=      L63.7
LD     L60.0
CALL   AXIS0_GOTO:SBR3, L63.7, X_Cmd_Pos:VD2000, X_Debug_Speed:VD2012, 0, X_Stop_Cmd:M20.2, #X_Teach_Done:L5.0, #X_Teach_Err:LB6, X_Curr_Pos_Scr:VD1900, X_Curr_Speed:MD4
Network 8
LD     X_Teach_EN:M18.7
A      #X_Teach_Done:L5.0
A      X_AXIS_INPOS:I1.4
R      X_Teach_EN:M18.7, 1
Network 9
// Y  Teaching...
LD     Y_Teach_EN:M19.0
=      L60.0
LD     Y_Teach_EN:M19.0
EU
=      L63.7
LD     L60.0
CALL   AXIS1_GOTO:SBR14, L63.7, Y_Cmd_Pos:VD2004, Y_Debug_Speed:VD2016, 0, Y_Stop_Cmd:M20.3, #Y_Teach_Done:L5.1, #Y_Teach_Err:LB7, Y_Curr_Pos_Scr:VD1904, Y_Curr_Speed:MD8
Network 10
LD     Y_Teach_EN:M19.0
A      #Y_Teach_Done:L5.1
A      Y_AXIS_INPOS:I1.7
R      Y_Teach_EN:M19.0, 1
Network 11
// Z  Teaching...
LD     Z_Teach_EN:M19.1
=      L60.0
LD     Z_Teach_EN:M19.1
EU
=      L63.7
LD     L60.0
CALL   AXIS2_GOTO:SBR25, L63.7, Z_Cmd_Pos:VD2008, Z_Debug_Speed:VD2020, 0, Z_Stop_Cmd:M20.4, #Z_Teach_Done:L5.2, #Z_Teach_Err:LB8, Z_Curr_Pos_Scr:VD1908, Z_Curr_Speed:MD12
Network 12
LD     Z_Teach_EN:M19.1
A      #Z_Teach_Done:L5.2
A      Z_AXIS_INPOS:I2.2
R      Z_Teach_EN:M19.1, 1
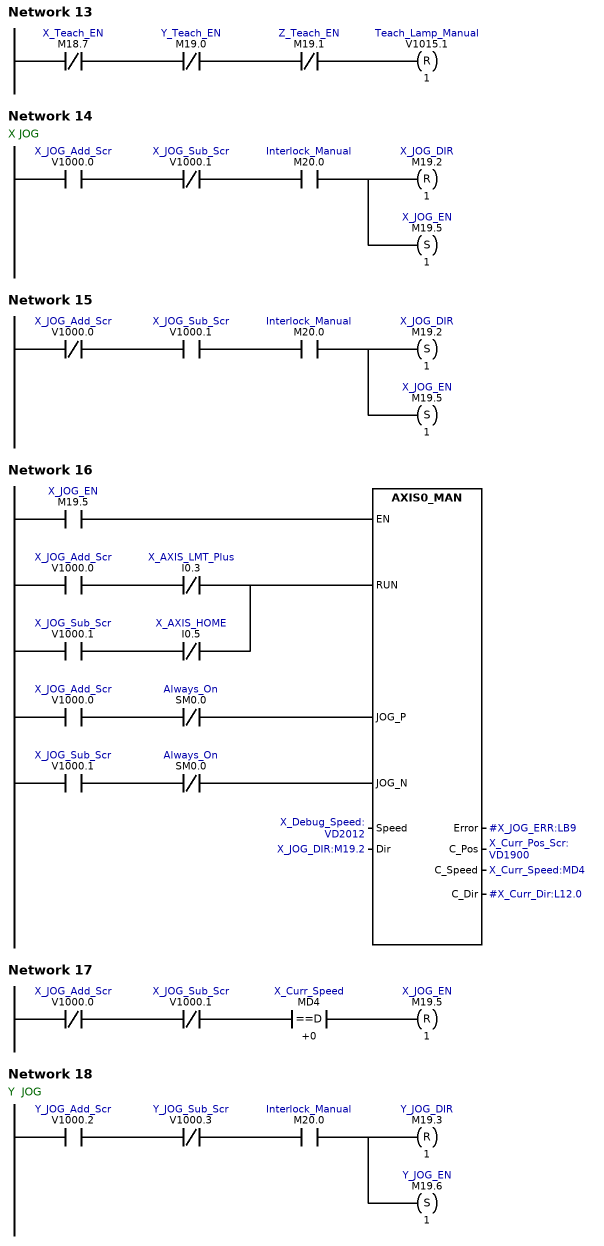
Network 13
LDN    X_Teach_EN:M18.7
AN     Y_Teach_EN:M19.0
AN     Z_Teach_EN:M19.1
R      Teach_Lamp_Manual:V1015.1, 1
Network 14
// X JOG
LD     X_JOG_Add_Scr:V1000.0
AN     X_JOG_Sub_Scr:V1000.1
A      Interlock_Manual:M20.0
R      X_JOG_DIR:M19.2, 1
S      X_JOG_EN:M19.5, 1
Network 15
LDN    X_JOG_Add_Scr:V1000.0
A      X_JOG_Sub_Scr:V1000.1
A      Interlock_Manual:M20.0
S      X_JOG_DIR:M19.2, 1
S      X_JOG_EN:M19.5, 1
Network 16
LD     X_JOG_EN:M19.5
=      L60.0
LD     X_JOG_Add_Scr:V1000.0
AN     X_AXIS_LMT_Plus:I0.3
LD     X_JOG_Sub_Scr:V1000.1
AN     X_AXIS_HOME:I0.5
OLD
=      L63.7
LD     X_JOG_Add_Scr:V1000.0
AN     Always_On:SM0.0
=      L63.6
LD     X_JOG_Sub_Scr:V1000.1
AN     Always_On:SM0.0
=      L63.5
LD     L60.0
CALL   AXIS0_MAN:SBR2, L63.7, L63.6, L63.5, X_Debug_Speed:VD2012, X_JOG_DIR:M19.2, #X_JOG_ERR:LB9, X_Curr_Pos_Scr:VD1900, X_Curr_Speed:MD4, #X_Curr_Dir:L12.0
Network 17
LDN    X_JOG_Add_Scr:V1000.0
AN     X_JOG_Sub_Scr:V1000.1
AD=    X_Curr_Speed:MD4, +0
R      X_JOG_EN:M19.5, 1
Network 18
// Y  JOG
LD     Y_JOG_Add_Scr:V1000.2
AN     Y_JOG_Sub_Scr:V1000.3
A      Interlock_Manual:M20.0
R      Y_JOG_DIR:M19.3, 1
S      Y_JOG_EN:M19.6, 1
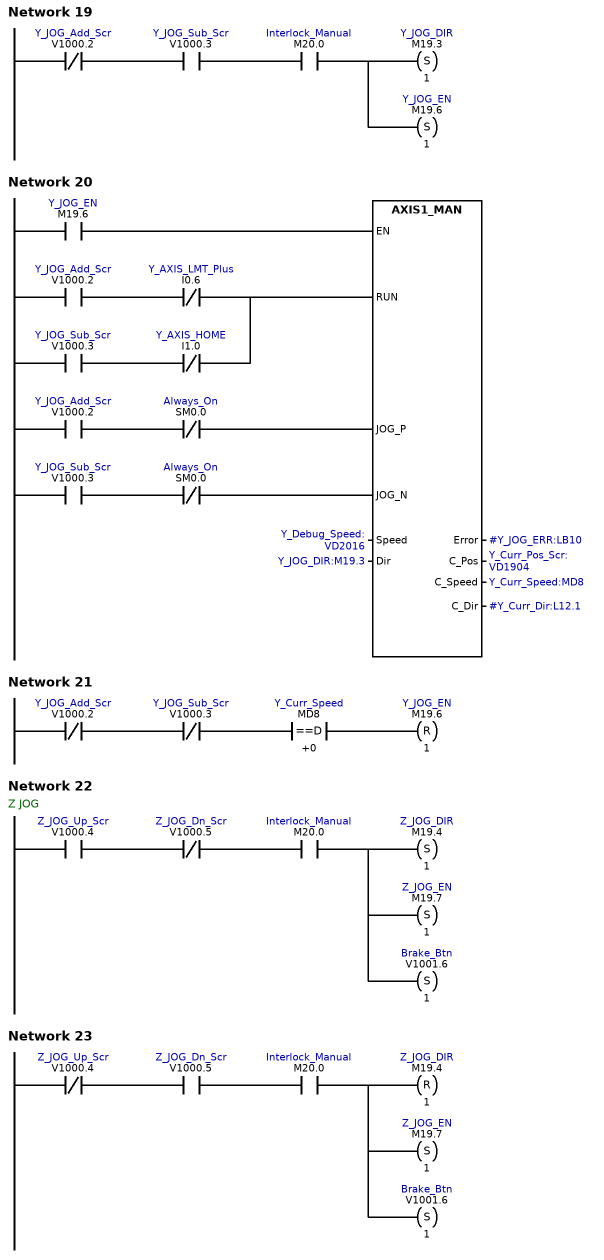
Network 19
LDN    Y_JOG_Add_Scr:V1000.2
A      Y_JOG_Sub_Scr:V1000.3
A      Interlock_Manual:M20.0
S      Y_JOG_DIR:M19.3, 1
S      Y_JOG_EN:M19.6, 1
Network 20
LD     Y_JOG_EN:M19.6
=      L60.0
LD     Y_JOG_Add_Scr:V1000.2
AN     Y_AXIS_LMT_Plus:I0.6
LD     Y_JOG_Sub_Scr:V1000.3
AN     Y_AXIS_HOME:I1.0
OLD
=      L63.7
LD     Y_JOG_Add_Scr:V1000.2
AN     Always_On:SM0.0
=      L63.6
LD     Y_JOG_Sub_Scr:V1000.3
AN     Always_On:SM0.0
=      L63.5
LD     L60.0
CALL   AXIS1_MAN:SBR13, L63.7, L63.6, L63.5, Y_Debug_Speed:VD2016, Y_JOG_DIR:M19.3, #Y_JOG_ERR:LB10, Y_Curr_Pos_Scr:VD1904, Y_Curr_Speed:MD8, #Y_Curr_Dir:L12.1
Network 21
LDN    Y_JOG_Add_Scr:V1000.2
AN     Y_JOG_Sub_Scr:V1000.3
AD=    Y_Curr_Speed:MD8, +0
R      Y_JOG_EN:M19.6, 1
Network 22
// Z JOG
LD     Z_JOG_Up_Scr:V1000.4
AN     Z_JOG_Dn_Scr:V1000.5
A      Interlock_Manual:M20.0
S      Z_JOG_DIR:M19.4, 1
S      Z_JOG_EN:M19.7, 1
S      Brake_Btn:V1001.6, 1
Network 23
LDN    Z_JOG_Up_Scr:V1000.4
A      Z_JOG_Dn_Scr:V1000.5
A      Interlock_Manual:M20.0
R      Z_JOG_DIR:M19.4, 1
S      Z_JOG_EN:M19.7, 1
S      Brake_Btn:V1001.6, 1
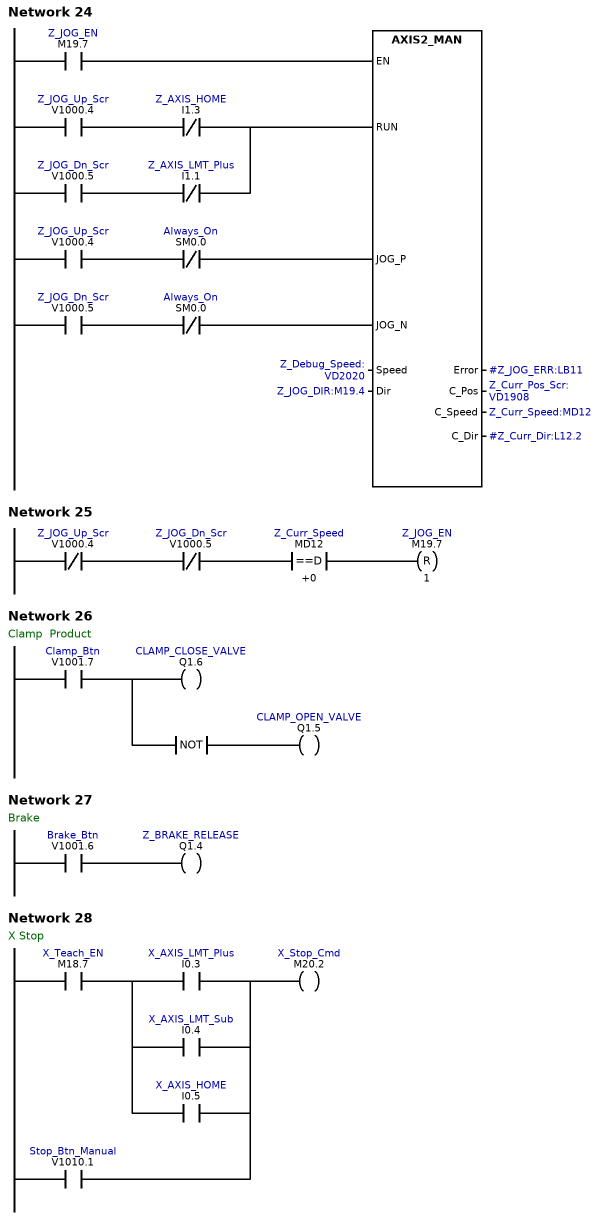
Network 24
LD     Z_JOG_EN:M19.7
=      L60.0
LD     Z_JOG_Up_Scr:V1000.4
AN     Z_AXIS_HOME:I1.3
LD     Z_JOG_Dn_Scr:V1000.5
AN     Z_AXIS_LMT_Plus:I1.1
OLD
=      L63.7
LD     Z_JOG_Up_Scr:V1000.4
AN     Always_On:SM0.0
=      L63.6
LD     Z_JOG_Dn_Scr:V1000.5
AN     Always_On:SM0.0
=      L63.5
LD     L60.0
CALL   AXIS2_MAN:SBR24, L63.7, L63.6, L63.5, Z_Debug_Speed:VD2020, Z_JOG_DIR:M19.4, #Z_JOG_ERR:LB11, Z_Curr_Pos_Scr:VD1908, Z_Curr_Speed:MD12, #Z_Curr_Dir:L12.2
Network 25
LDN    Z_JOG_Up_Scr:V1000.4
AN     Z_JOG_Dn_Scr:V1000.5
AD=    Z_Curr_Speed:MD12, +0
R      Z_JOG_EN:M19.7, 1
Network 26
// Clamp  Product
LD     Clamp_Btn:V1001.7
=      CLAMP_CLOSE_VALVE:Q1.6
NOT
=      CLAMP_OPEN_VALVE:Q1.5
Network 27
// Brake
LD     Brake_Btn:V1001.6
=      Z_BRAKE_RELEASE:Q1.4
Network 28
// X Stop
LD     X_Teach_EN:M18.7
LD     X_AXIS_LMT_Plus:I0.3
O      X_AXIS_LMT_Sub:I0.4
O      X_AXIS_HOME:I0.5
ALD
O      Stop_Btn_Manual:V1010.1
=      X_Stop_Cmd:M20.2
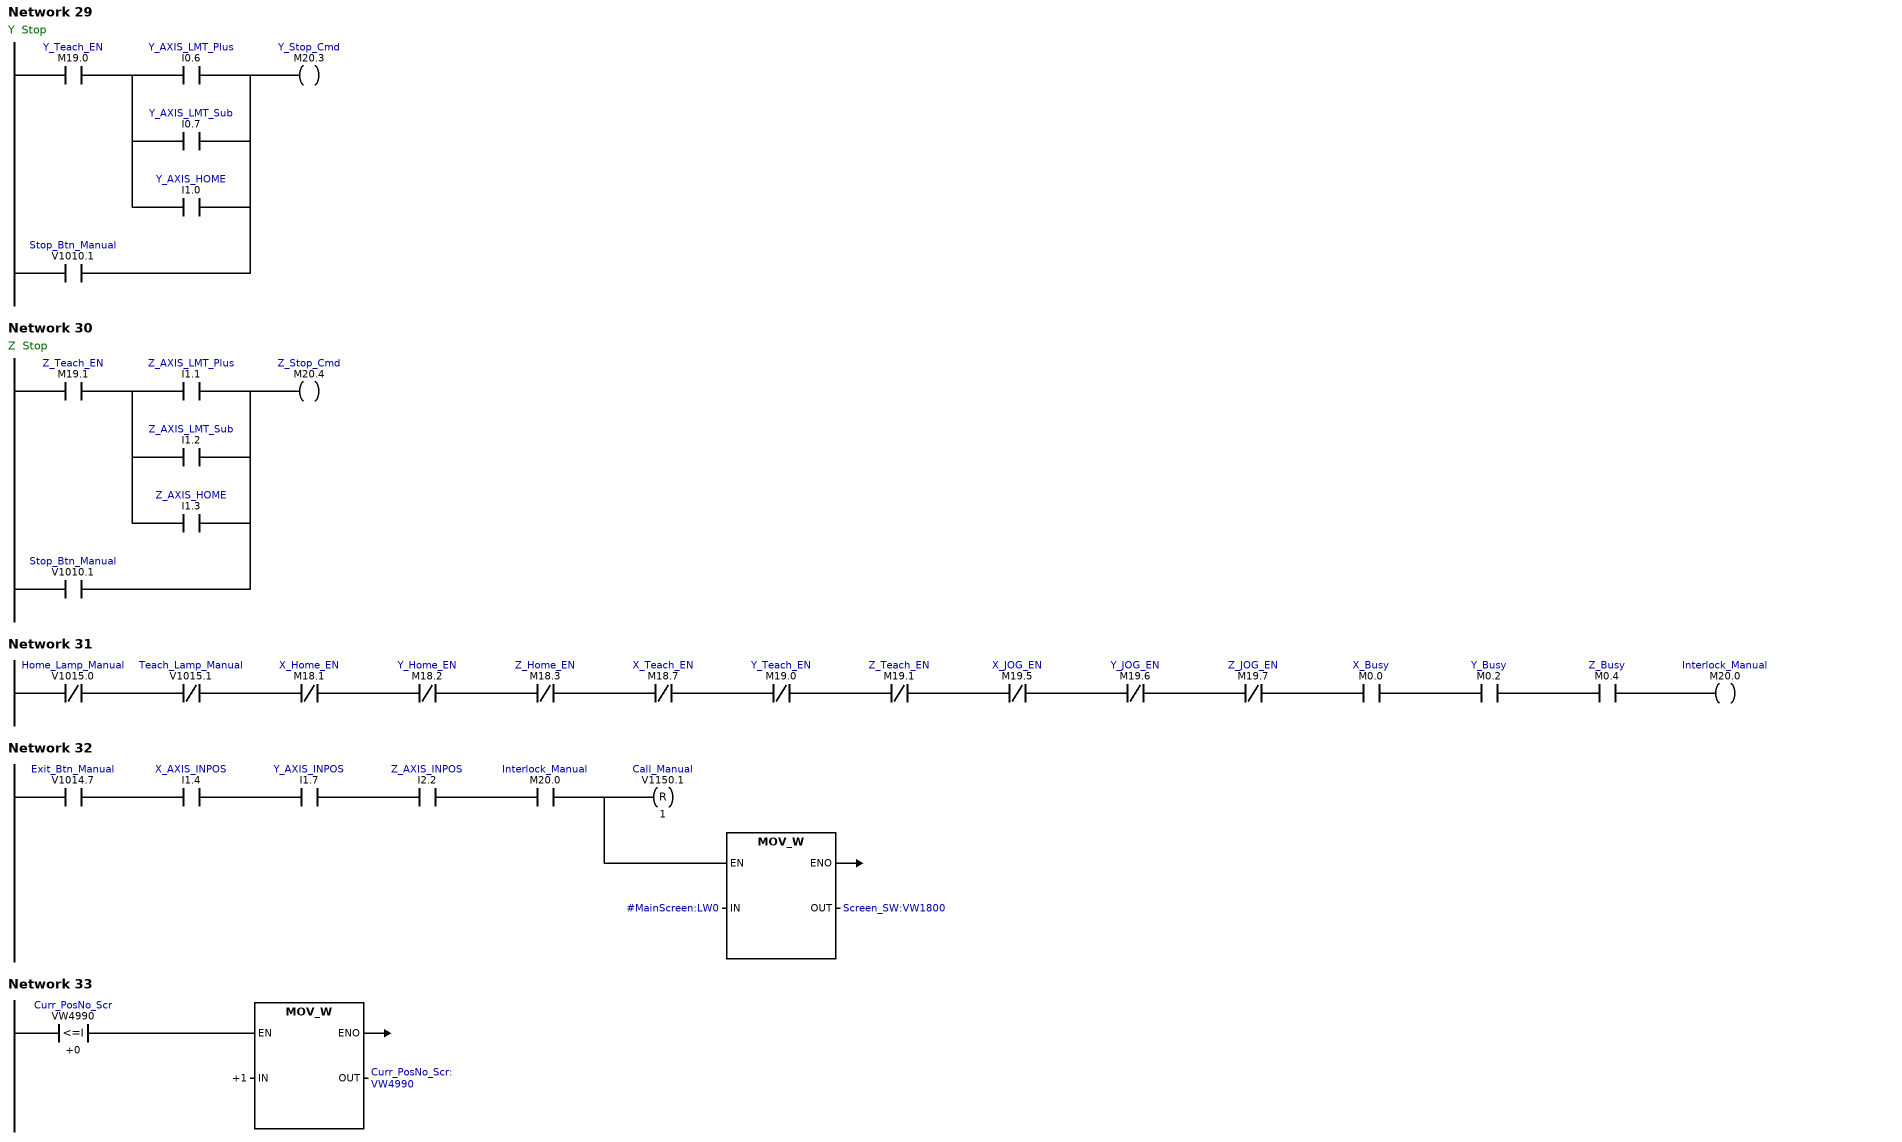
Network 29
// Y  Stop
LD     Y_Teach_EN:M19.0
LD     Y_AXIS_LMT_Plus:I0.6
O      Y_AXIS_LMT_Sub:I0.7
O      Y_AXIS_HOME:I1.0
ALD
O      Stop_Btn_Manual:V1010.1
=      Y_Stop_Cmd:M20.3
Network 30
// Z  Stop
LD     Z_Teach_EN:M19.1
LD     Z_AXIS_LMT_Plus:I1.1
O      Z_AXIS_LMT_Sub:I1.2
O      Z_AXIS_HOME:I1.3
ALD
O      Stop_Btn_Manual:V1010.1
=      Z_Stop_Cmd:M20.4
Network 31
LDN    Home_Lamp_Manual:V1015.0
AN     Teach_Lamp_Manual:V1015.1
AN     X_Home_EN:M18.1
AN     Y_Home_EN:M18.2
AN     Z_Home_EN:M18.3
AN     X_Teach_EN:M18.7
AN     Y_Teach_EN:M19.0
AN     Z_Teach_EN:M19.1
AN     X_JOG_EN:M19.5
AN     Y_JOG_EN:M19.6
AN     Z_JOG_EN:M19.7
A      X_Busy:M0.0
A      Y_Busy:M0.2
A      Z_Busy:M0.4
=      Interlock_Manual:M20.0
Network 32
LD     Exit_Btn_Manual:V1014.7
A      X_AXIS_INPOS:I1.4
A      Y_AXIS_INPOS:I1.7
A      Z_AXIS_INPOS:I2.2
A      Interlock_Manual:M20.0
R      Call_Manual:V1150.1, 1
MOVW   #MainScreen:LW0, Screen_SW:VW1800
Network 33
LDW<=  Curr_PosNo_Scr:VW4990, +0
MOVW   +1, Curr_PosNo_Scr:VW4990
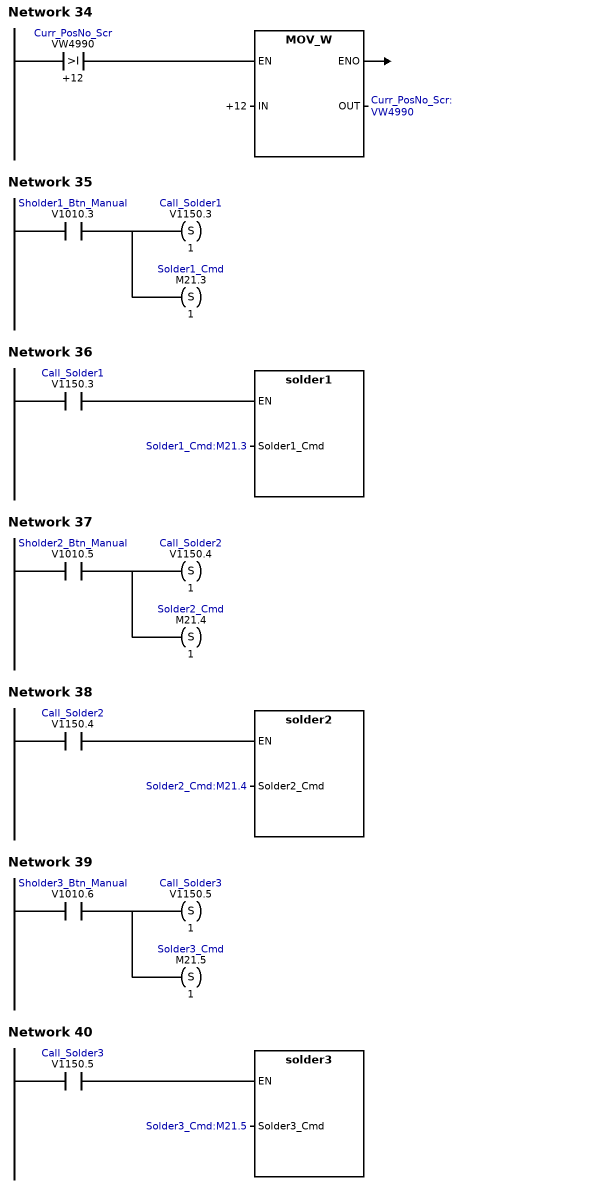
Network 34
LDW>   Curr_PosNo_Scr:VW4990, +12
MOVW   +12, Curr_PosNo_Scr:VW4990
Network 35
LD     Sholder1_Btn_Manual:V1010.3
S      Call_Solder1:V1150.3, 1
S      Solder1_Cmd:M21.3, 1
Network 36
LD     Call_Solder1:V1150.3
CALL   solder1:SBR38, Solder1_Cmd:M21.3
Network 37
LD     Sholder2_Btn_Manual:V1010.5
S      Call_Solder2:V1150.4, 1
S      Solder2_Cmd:M21.4, 1
Network 38
LD     Call_Solder2:V1150.4
CALL   solder2:SBR39, Solder2_Cmd:M21.4
Network 39
LD     Sholder3_Btn_Manual:V1010.6
S      Call_Solder3:V1150.5, 1
S      Solder3_Cmd:M21.5, 1
Network 40
LD     Call_Solder3:V1150.5
CALL   solder3:SBR40, Solder3_Cmd:M21.5
END_SUBROUTINE_BLOCK

// SBR1: protected block, not included

// SBR2: protected block, not included

// SBR3: protected block, not included

// SBR4: protected block, not included

// SBR5: protected block, not included

// SBR6: protected block, not included

// SBR7: protected block, not included

// SBR8: protected block, not included

// SBR9: protected block, not included

// SBR10: protected block, not included

// SBR11: protected block, not included

// SBR12: protected block, not included

// SBR13: protected block, not included

// SBR14: protected block, not included

// SBR15: protected block, not included

// SBR16: protected block, not included

// SBR17: protected block, not included

// SBR18: protected block, not included

// SBR19: protected block, not included

// SBR20: protected block, not included

// SBR21: protected block, not included

// SBR22: protected block, not included

// SBR23: protected block, not included

// SBR24: protected block, not included

// SBR25: protected block, not included

// SBR26: protected block, not included

// SBR27: protected block, not included

// SBR28: protected block, not included

// SBR29: protected block, not included

// SBR30: protected block, not included

// SBR31: protected block, not included

// SBR32: protected block, not included

// SBR33: protected block, not included

SUBROUTINE_BLOCK Auto:SBR34
TITLE=子例程注释
VAR
Z_Up_Done:BOOL;	// L0.0 
X_Run_Done:BOOL;	// L0.1 
Y_Run_Done:BOOL;	// L0.2 
Z_Run_Done:BOOL;	// L0.3 
END_VAR
BEGIN
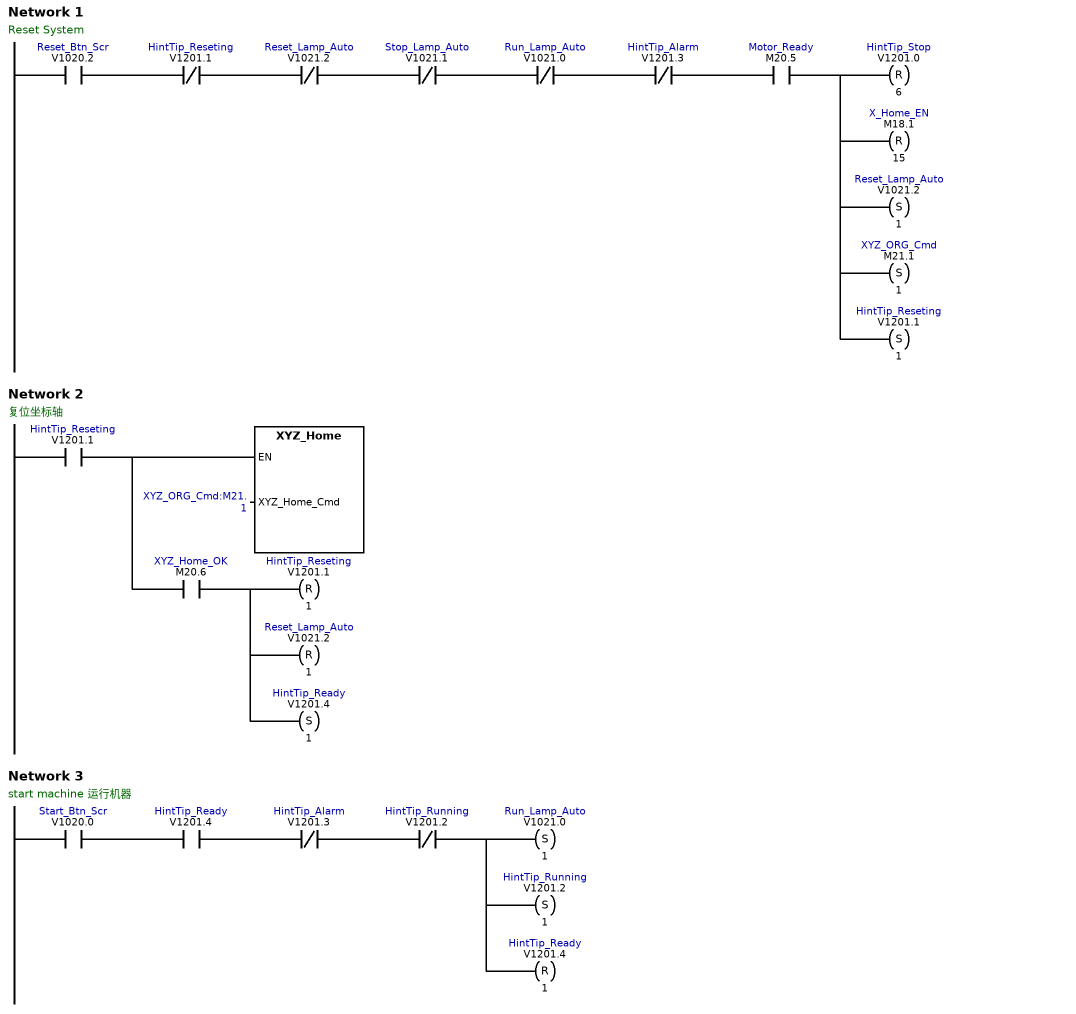
Network 1
// Reset System
LD     Reset_Btn_Scr:V1020.2
AN     HintTip_Reseting:V1201.1
AN     Reset_Lamp_Auto:V1021.2
AN     Stop_Lamp_Auto:V1021.1
AN     Run_Lamp_Auto:V1021.0
AN     HintTip_Alarm:V1201.3
A      Motor_Ready:M20.5
R      HintTip_Stop:V1201.0, 6
R      X_Home_EN:M18.1, 15
S      Reset_Lamp_Auto:V1021.2, 1
S      XYZ_ORG_Cmd:M21.1, 1
S      HintTip_Reseting:V1201.1, 1
Network 2
// 复位坐标轴
LD     HintTip_Reseting:V1201.1
CALL   XYZ_Home:SBR37, XYZ_ORG_Cmd:M21.1
A      XYZ_Home_OK:M20.6
R      HintTip_Reseting:V1201.1, 1
R      Reset_Lamp_Auto:V1021.2, 1
S      HintTip_Ready:V1201.4, 1
Network 3
// start machine 运行机器
LD     Start_Btn_Scr:V1020.0
A      HintTip_Ready:V1201.4
AN     HintTip_Alarm:V1201.3
AN     HintTip_Running:V1201.2
S      Run_Lamp_Auto:V1021.0, 1
S      HintTip_Running:V1201.2, 1
R      HintTip_Ready:V1201.4, 1
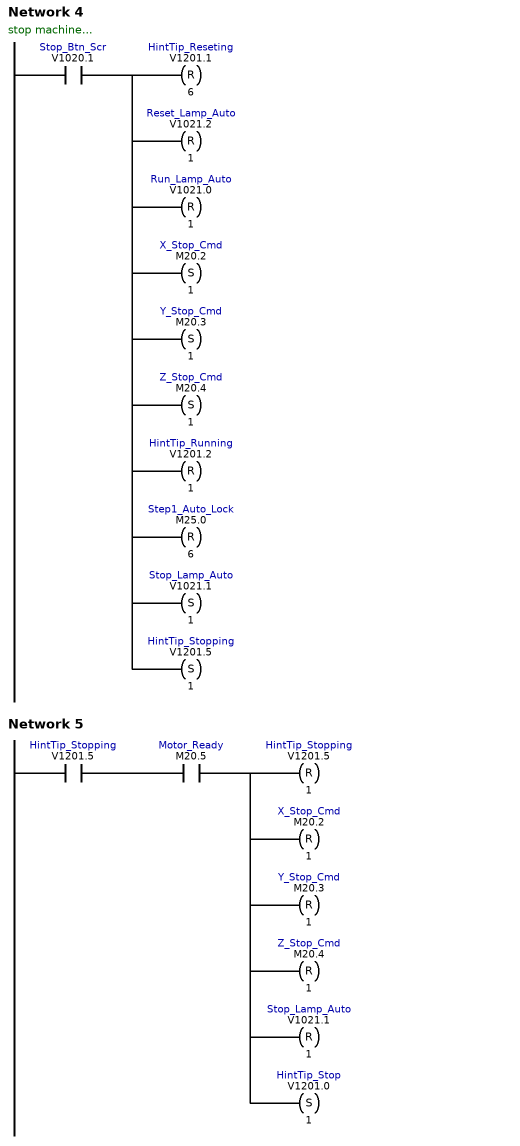
Network 4
// stop machine...
LD     Stop_Btn_Scr:V1020.1
R      HintTip_Reseting:V1201.1, 6
R      Reset_Lamp_Auto:V1021.2, 1
R      Run_Lamp_Auto:V1021.0, 1
S      X_Stop_Cmd:M20.2, 1
S      Y_Stop_Cmd:M20.3, 1
S      Z_Stop_Cmd:M20.4, 1
R      HintTip_Running:V1201.2, 1
R      Step1_Auto_Lock:M25.0, 6
S      Stop_Lamp_Auto:V1021.1, 1
S      HintTip_Stopping:V1201.5, 1
Network 5
LD     HintTip_Stopping:V1201.5
A      Motor_Ready:M20.5
R      HintTip_Stopping:V1201.5, 1
R      X_Stop_Cmd:M20.2, 1
R      Y_Stop_Cmd:M20.3, 1
R      Z_Stop_Cmd:M20.4, 1
R      Stop_Lamp_Auto:V1021.1, 1
S      HintTip_Stop:V1201.0, 1
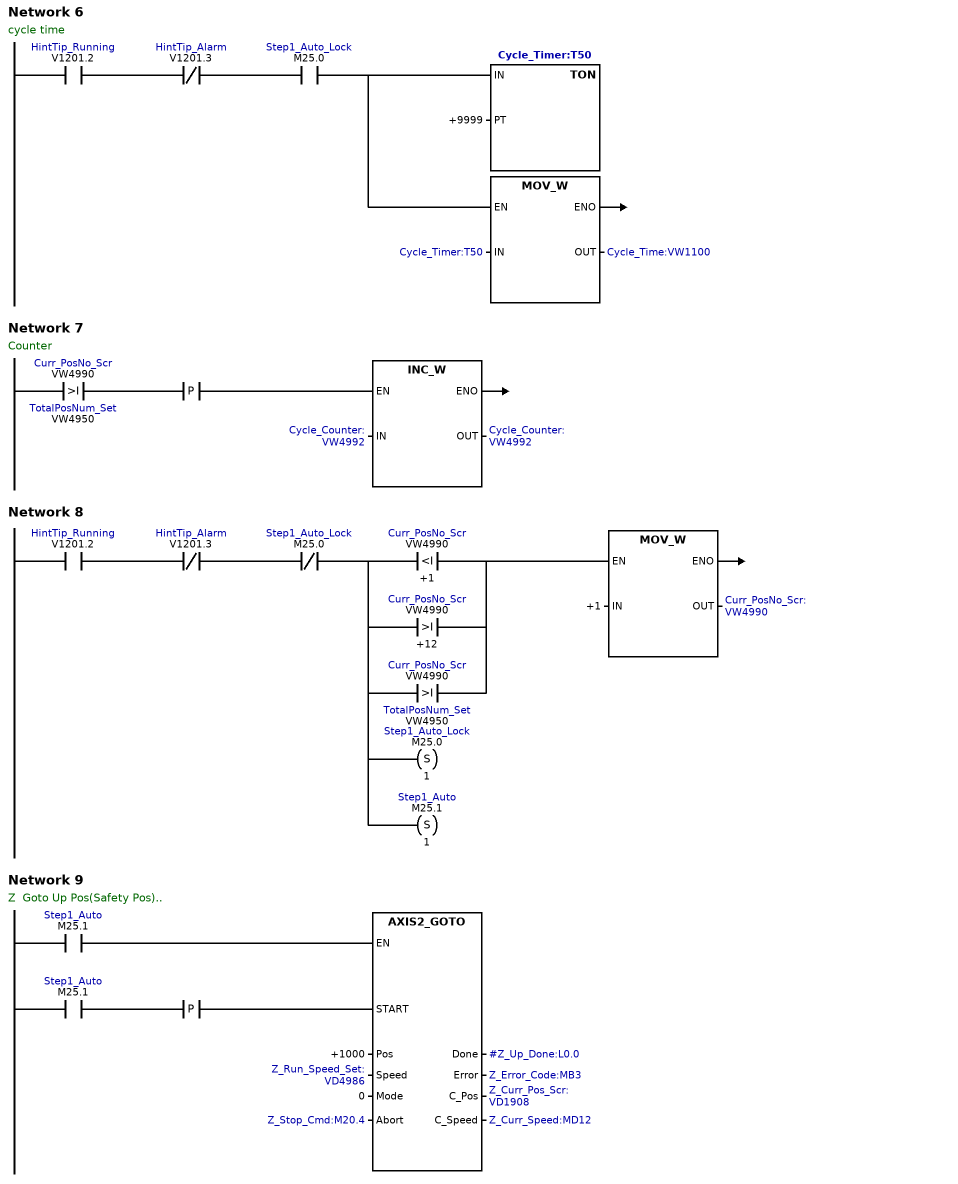
Network 6
// cycle time
LD     HintTip_Running:V1201.2
AN     HintTip_Alarm:V1201.3
A      Step1_Auto_Lock:M25.0
TON    Cycle_Timer:T50, +9999
MOVW   Cycle_Timer:T50, Cycle_Time:VW1100
Network 7
// Counter
LDW>   Curr_PosNo_Scr:VW4990, TotalPosNum_Set:VW4950
EU
INCW   Cycle_Counter:VW4992
Network 8
LD     HintTip_Running:V1201.2
AN     HintTip_Alarm:V1201.3
AN     Step1_Auto_Lock:M25.0
LPS
LDW<   Curr_PosNo_Scr:VW4990, +1
OW>    Curr_PosNo_Scr:VW4990, +12
OW>    Curr_PosNo_Scr:VW4990, TotalPosNum_Set:VW4950
ALD
MOVW   +1, Curr_PosNo_Scr:VW4990
LPP
S      Step1_Auto_Lock:M25.0, 1
S      Step1_Auto:M25.1, 1
Network 9
// Z  Goto Up Pos(Safety Pos)..
LD     Step1_Auto:M25.1
=      L60.0
LD     Step1_Auto:M25.1
EU
=      L63.7
LD     L60.0
CALL   AXIS2_GOTO:SBR25, L63.7, +1000, Z_Run_Speed_Set:VD4986, 0, Z_Stop_Cmd:M20.4, #Z_Up_Done:L0.0, Z_Error_Code:MB3, Z_Curr_Pos_Scr:VD1908, Z_Curr_Speed:MD12
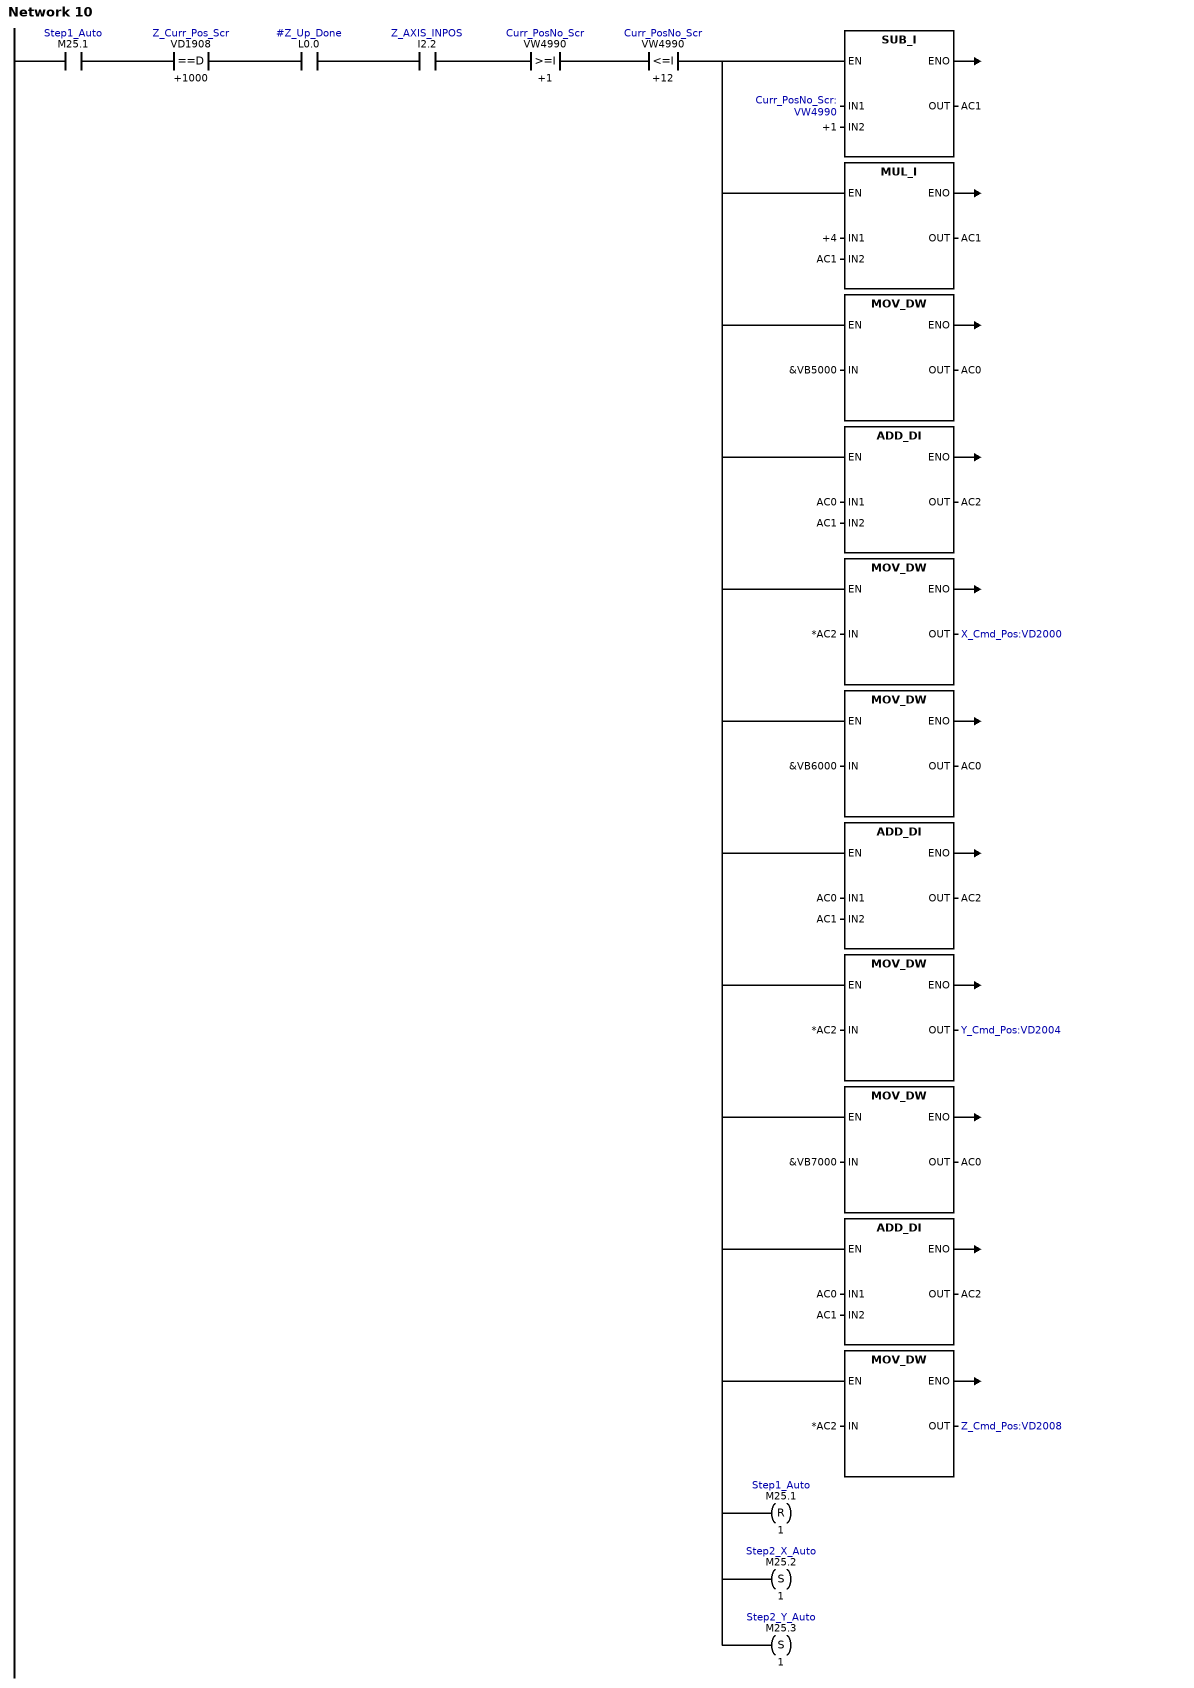
Network 10
LD     Step1_Auto:M25.1
AD=    Z_Curr_Pos_Scr:VD1908, +1000
A      #Z_Up_Done:L0.0
A      Z_AXIS_INPOS:I2.2
AW>=   Curr_PosNo_Scr:VW4990, +1
AW<=   Curr_PosNo_Scr:VW4990, +12
MOVW   Curr_PosNo_Scr:VW4990, AC1
-I     +1, AC1
*I     +4, AC1
MOVD   &VB5000, AC0
MOVD   AC0, AC2
+D     AC1, AC2
MOVD   *AC2, X_Cmd_Pos:VD2000
MOVD   &VB6000, AC0
MOVD   AC0, AC2
+D     AC1, AC2
MOVD   *AC2, Y_Cmd_Pos:VD2004
MOVD   &VB7000, AC0
MOVD   AC0, AC2
+D     AC1, AC2
MOVD   *AC2, Z_Cmd_Pos:VD2008
R      Step1_Auto:M25.1, 1
S      Step2_X_Auto:M25.2, 1
S      Step2_Y_Auto:M25.3, 1
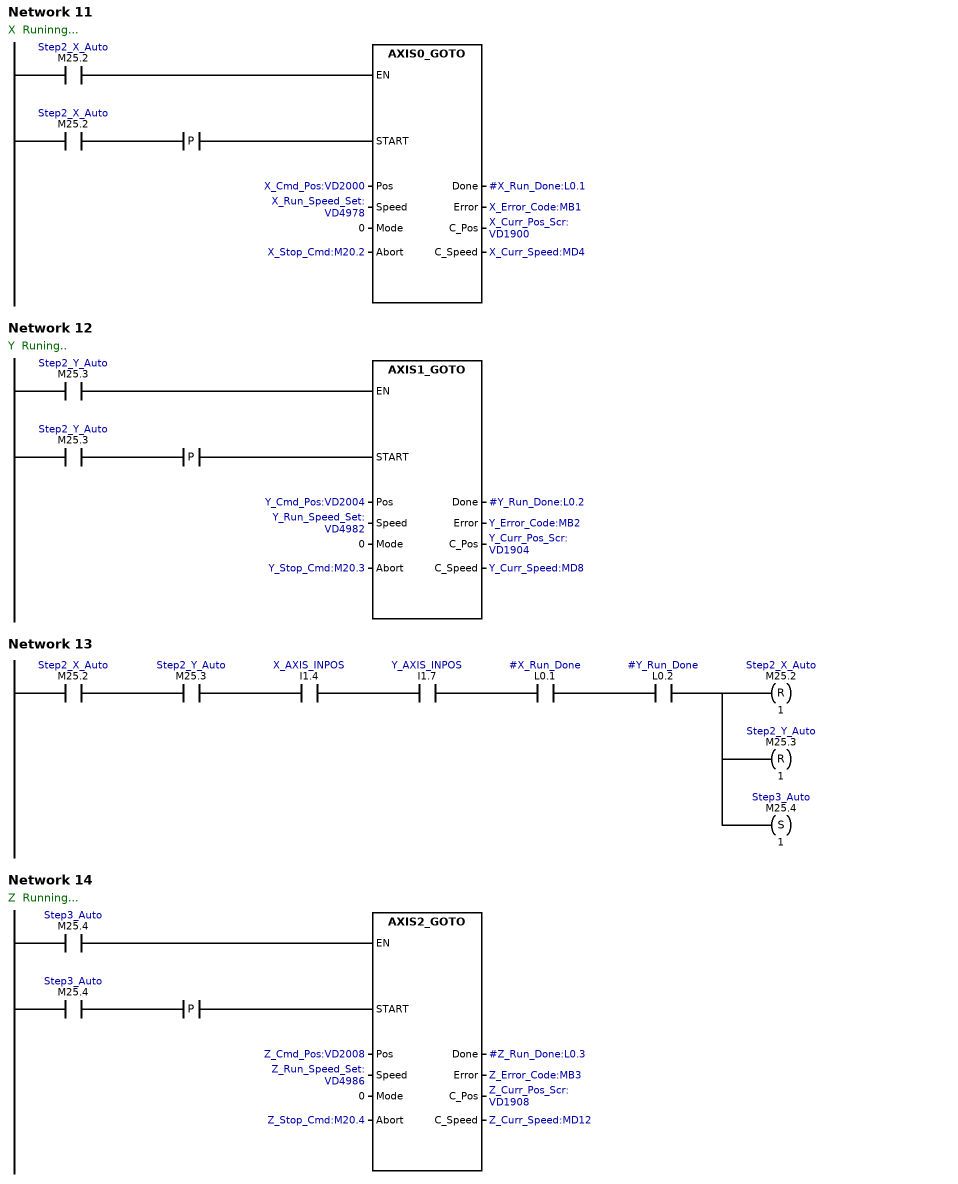
Network 11
// X  Runinng...
LD     Step2_X_Auto:M25.2
=      L60.0
LD     Step2_X_Auto:M25.2
EU
=      L63.7
LD     L60.0
CALL   AXIS0_GOTO:SBR3, L63.7, X_Cmd_Pos:VD2000, X_Run_Speed_Set:VD4978, 0, X_Stop_Cmd:M20.2, #X_Run_Done:L0.1, X_Error_Code:MB1, X_Curr_Pos_Scr:VD1900, X_Curr_Speed:MD4
Network 12
// Y  Runing..
LD     Step2_Y_Auto:M25.3
=      L60.0
LD     Step2_Y_Auto:M25.3
EU
=      L63.7
LD     L60.0
CALL   AXIS1_GOTO:SBR14, L63.7, Y_Cmd_Pos:VD2004, Y_Run_Speed_Set:VD4982, 0, Y_Stop_Cmd:M20.3, #Y_Run_Done:L0.2, Y_Error_Code:MB2, Y_Curr_Pos_Scr:VD1904, Y_Curr_Speed:MD8
Network 13
LD     Step2_X_Auto:M25.2
A      Step2_Y_Auto:M25.3
A      X_AXIS_INPOS:I1.4
A      Y_AXIS_INPOS:I1.7
A      #X_Run_Done:L0.1
A      #Y_Run_Done:L0.2
R      Step2_X_Auto:M25.2, 1
R      Step2_Y_Auto:M25.3, 1
S      Step3_Auto:M25.4, 1
Network 14
// Z  Running...
LD     Step3_Auto:M25.4
=      L60.0
LD     Step3_Auto:M25.4
EU
=      L63.7
LD     L60.0
CALL   AXIS2_GOTO:SBR25, L63.7, Z_Cmd_Pos:VD2008, Z_Run_Speed_Set:VD4986, 0, Z_Stop_Cmd:M20.4, #Z_Run_Done:L0.3, Z_Error_Code:MB3, Z_Curr_Pos_Scr:VD1908, Z_Curr_Speed:MD12
